// Register module to system
pModuleDef := ISystemBase.regModule(pAdsInfo:=ADR(sC_Ads_Info), pMapInfo:=ADR(sMappingInfo));
IF pModuleDef = 0 THEN RETURN; END_IF

// Command / Status interface
PRG_SYSTEMBASE.getSystemStatusInterface(iSystemStatus=>iSystemStatus);
PRG_SYSTEMBASE.getSystemCmdInterface(iSystemCmd=>iSystemCmd);

// Let the sleep be handled by the library
iSystemCmd.registerPucSleepInterface(pCmd_Sleep:=ADR(sADS_Machine[1].sI_Sleep),
                                     pCmd_WakeUp:=ADR(sADS_Machine[1].sI_WakeUp));

// Get Task cycle information
Fb_GetCurTskIndx();
tskL_ActTaskInfo := _TaskInfo[FB_GetCurTskIndx.index];
lL_TaskCycleTime := UDINT_TO_REAL(tskL_ActTaskInfo.CycleTime) / 10_000_000.0;

(* -- Messages ----------------------------------------------------------------------------------*)
initMsg();


(*************************************************************************************************)
(*Function Blocks Init*)
(*************************************************************************************************)
(*Cleaning station*)
(*Module 1*)
sADS_CleanProcess[1].aO_Name                  := 'Clean Process M2';
sADS_CleanProcess[1].bO_AxisProcessMovingVisible := FALSE;
//Clean unit
sADS_CleanAxis[1].aO_Name                     := 'M2: CU-Axis [mm]';
sADS_CleanAxis[1].sO_AxisPosition.fC_Min      := 0;    (*Value is used for display of axes at PUC*)
sADS_CleanAxis[1].sO_AxisPosition.fC_Max      := 586.0;
fb_CleaningCU[1].pC_MsgInterface              := ADR(sADS_CleanAxis[1].sO_Message);
fb_CleaningCU[1].iC_BlockId                   := eMa_BLK_CLEANAXIS;
fb_CleaningCU[1].fB_Axis.fI_Tolerance         := 0.001;
fb_CleaningCU[1].fB_Axis.fI_PosControllerGain := 5;
fb_CleaningCU[1].fB_Axis.fI_Axis_Scaling      := (0.1512 * 1/10);
fb_CleaningCU[1].fB_Axis.fI_SetPositionValue  := -0.01;				(*Reference sensor is at -10mm*)
fb_CleaningCU[1].fB_Axis.fI_EncoderScaling    := 1048576			(*262.144 * 4*);

//Clean head
sADS_CleanAxis[2].aO_Name                     := 'M2: CH-Axis [mm]';
sADS_CleanAxis[2].sO_AxisPosition.fC_Min      := -1;
sADS_CleanAxis[2].sO_AxisPosition.fC_Max      := 400.0;
fb_CleaningCH[1].pC_MsgInterface              := ADR(sADS_CleanAxis[2].sO_Message);
fb_CleaningCH[1].iC_BlockId                   := eMa_BLK_CLEANAXIS;
fb_CleaningCH[1].fB_Axis.fI_Tolerance         := 0.001;
fb_CleaningCH[1].fB_Axis.fI_PosControllerGain := 5;
fb_CleaningCH[1].fB_Axis.fI_Axis_Scaling      := (0.010 * 1/10);
fb_CleaningCH[1].fB_Axis.fI_SetPositionValue  := -0.001;      (*Reference sensor is at -1mm*)
fb_CleaningCH[1].fB_Axis.fI_EncoderScaling    := 1048576			(*262.144 * 4*);

//Print unit
sADS_CleanAxis[3].aO_Name                     := 'M2: PU-Axis [mm]';
sADS_CleanAxis[3].sO_AxisPosition.fC_Min      := 0.5;  (********(Köbi) Korrektur 0.5 statt 1 *)
sADS_CleanAxis[3].sO_AxisPosition.fC_Max      := 250;
fb_CleaningPU[1].pC_MsgInterface              := ADR(sADS_CleanAxis[3].sO_Message);
fb_CleaningPU[1].iC_BlockId                   := eMa_BLK_CLEANAXIS;
fb_CleaningPU[1].fB_Axis.fI_Tolerance         := 0.0001;
fb_CleaningPU[1].fB_Axis.fI_PosControllerGain := 10;
fb_CleaningPU[1].fB_Axis.fI_Axis_Scaling      := 0.001; (******(Köbi) Korrektur Ration 0.001 statt ...*) //0.016 / 50 * 3;	(*Steigung Spindel / Übersetzung * Winkelgetriebe*)
fb_CleaningPU[1].fB_Axis.fI_SetPositionValue  := 0.010;           (*Calibrate manually at 10mm*)
fb_CleaningPU[1].fB_Axis.fI_EncoderScaling    := 1048576			(*65536*);

//Ink interface
sADS_CleanAxis[4].sO_AxisPosition.fC_Min      := 0;     (*Dummy*)
sADS_CleanAxis[4].sO_AxisPosition.fC_Max      := 1000;  (*Dummy*)


(*Module 2*)
sADS_CleanProcess[2].aO_Name                  := 'Clean Process M3';
sADS_CleanProcess[2].bO_AxisProcessMovingVisible := FALSE;
//Clean unit
sADS_CleanAxis[5].aO_Name                     := 'M3: CU-Axis [mm]';
sADS_CleanAxis[5].sO_AxisPosition.fC_Min      := 0;    (*Value is used for display of axes at PUC*)
sADS_CleanAxis[5].sO_AxisPosition.fC_Max      := 586.0;
fb_CleaningCU[2].pC_MsgInterface              := ADR(sADS_CleanAxis[5].sO_Message);
fb_CleaningCU[2].iC_BlockId                   := eMa_BLK_CLEANAXIS;
fb_CleaningCU[2].fB_Axis.fI_Tolerance         := 0.001;
fb_CleaningCU[2].fB_Axis.fI_PosControllerGain := 5;
fb_CleaningCU[2].fB_Axis.fI_Axis_Scaling      := (0.1512 * 1/10);
fb_CleaningCU[2].fB_Axis.fI_SetPositionValue  := -0.01;				(*Reference sensor is at -10mm*)
fb_CleaningCU[2].fB_Axis.fI_EncoderScaling    := 1048576			(*262.144 * 4*);

//Clean head
sADS_CleanAxis[6].aO_Name                     := 'M3: CH-Axis [mm]';
sADS_CleanAxis[6].sO_AxisPosition.fC_Min      := -1;
sADS_CleanAxis[6].sO_AxisPosition.fC_Max      := 400.0;
fb_CleaningCH[2].pC_MsgInterface              := ADR(sADS_CleanAxis[6].sO_Message);
fb_CleaningCH[2].iC_BlockId                   := eMa_BLK_CLEANAXIS;
fb_CleaningCH[2].fB_Axis.fI_Tolerance         := 0.001;
fb_CleaningCH[2].fB_Axis.fI_PosControllerGain := 5;
fb_CleaningCH[2].fB_Axis.fI_Axis_Scaling      := (0.010 * 1/10);
fb_CleaningCH[2].fB_Axis.fI_SetPositionValue  := -0.001;      (*Reference sensor is at -1mm*)
fb_CleaningCH[2].fB_Axis.fI_EncoderScaling    := 1048576			(*262.144 * 4*);

//Print unit
sADS_CleanAxis[7].aO_Name                     := 'M3: PU-Axis [mm]';
sADS_CleanAxis[7].sO_AxisPosition.fC_Min      := 0.5;  (********(Köbi) Korrektur 0.5 statt 1 *)
sADS_CleanAxis[7].sO_AxisPosition.fC_Max      := 250;
fb_CleaningPU[2].pC_MsgInterface              := ADR(sADS_CleanAxis[7].sO_Message);
fb_CleaningPU[2].iC_BlockId                   := eMa_BLK_CLEANAXIS;
fb_CleaningPU[2].fB_Axis.fI_Tolerance         := 0.0001;
fb_CleaningPU[2].fB_Axis.fI_PosControllerGain := 10;
fb_CleaningPU[2].fB_Axis.fI_Axis_Scaling      := 0.001; (******(Köbi) Korrektur Ration 0.001 statt ...*) //0.016 / 50 * 3;	(*Steigung Spindel / Übersetzung * Winkelgetriebe*)
fb_CleaningPU[2].fB_Axis.fI_SetPositionValue  := 0.010;            (*Calibrate manually at 10mm*)
fb_CleaningPU[2].fB_Axis.fI_EncoderScaling    := 1048576			(*65536*);

//Ink interface
sADS_CleanAxis[8].sO_AxisPosition.fC_Min      := 0;     (*Dummy*)
sADS_CleanAxis[8].sO_AxisPosition.fC_Max      := 1000;  (*Dummy*)

//Link reference to machine base
//X: clean unit
//Y: clean head
//Z: print unit
FOR iL_Counter := 1 TO iCMa_NB_Cp DO
  fb_CleanProcess     [iL_Counter].I_MachineStatus := fb_Machine;
  fb_CleaningCU       [iL_Counter].I_MachineStatus := fb_Machine;
  fb_CleaningPU       [iL_Counter].I_MachineStatus := fb_Machine;
  fb_CleaningCH       [iL_Counter].I_MachineStatus := fb_Machine;
  fb_CleaningValvePump[iL_Counter].I_MachineStatus := fb_Machine;
  
  //Init blocks
  fb_CleanProcess[iL_Counter].pC_MsgInterface := ADR(sADS_CleanProcess[iL_Counter].sO_Message);
  fb_CleanProcess[iL_Counter].iC_BlockId      := eMa_BLK_CLEANPROC;
  
  fb_CleanProcess     [iL_Counter].mInit();
  fb_CleaningCU       [iL_Counter].mInit();
  fb_CleaningPU       [iL_Counter].mInit();
  fb_CleaningCH       [iL_Counter].mInit();
  fb_CleaningValvePump[iL_Counter].mInit();
  
  //Register cleaning devices
  fb_CleanProcess[iL_Counter].mRegisterDevice(fb_CleaningCU[iL_Counter]);
  fb_CleanProcess[iL_Counter].mRegisterDevice(fb_CleaningPU[iL_Counter]);
  fb_CleanProcess[iL_Counter].mRegisterDevice(fb_CleaningCH[iL_Counter]);
  fb_CleanProcess[iL_Counter].mRegisterDevice(fb_CleaningValvePump[iL_Counter]);

  fb_MotionInterlock[iL_Counter].fCCU_SafePosition[1]      := 0.005;
  fb_MotionInterlock[iL_Counter].fCCU_SafePosition[2]      := 0.584;
  fb_MotionInterlock[iL_Counter].fCCU_SafePosition[3]      := 0.586;
  fb_MotionInterlock[iL_Counter].fCPU_SafePosition[1]      := 0.160;
  fb_MotionInterlock[iL_Counter].fCPU_SafePosition[2]      := 0.165;
  fb_MotionInterlock[iL_Counter].fCCU_CleaningPosition     := 0.584;
  fb_MotionInterlock[iL_Counter].fCCU_Tolerance            := 0.002;
  fb_MotionInterlock[iL_Counter].fCPU_Tolerance            := 0.0005;
END_FOR;

(* -- Mapping -----------------------------------------------------------------------------------*)
Mapping();

(* -- Recipe ------------------------------------------------------------------------------------*)
pFbRecipeMngr := PRG_SYSTEMBASE.registerRecipe(
  aI_RecipePath           := CONCAT(aC_PlcConfigPath, aC_PlcRecipeSubPath),
  aI_RecipeDefinitionName := sC_Ads_Info.aType  (*is set in Mapping*)
);

(* -- BlockId saving ----------------------------------------------------------------------------*)
PRG_SYSTEMBASE.fbBlockIdSave.registerModule(
  aI_StoragePath := CONCAT(aC_PlcConfigPath, aC_PlcBlockIdSubPath),
  pI_Ads_Info    := ADR(sC_Ads_Info)
);

bL_RemVar_Init := TRUE;    (* Write variables by remanent variables *)
RemVar();

// init finished
bO_InitOk :=  TRUE;
END_METHOD

METHOD PRIVATE initMsg

(*Machine messaging*)
sL_MsgConfigMachine[1].bI_Enable                  := TRUE;
sL_MsgConfigMachine[1].pI_FbMsgHandler            := ADR(fb_MachineMsgHandler[1]);

fb_MachineMsgHandler[1].pI_MsgQueue               := ADR(fb_MsgQueueMachine[1]);

fb_MsgQueueMachine[1].pI_MsgInterface             := ADR(sADS_Machine[1].sO_Message);
fb_MsgQueueMachine[1].cI_MaxElement               := 5;

FOR iL_Counter := 1 TO iCMa_NB_MSG DO
  fb_MachineMsg[1, iL_Counter].pI_MsgConfig       := ADR(sL_MsgConfigMachine[1]);
  fb_MachineMsg[1, iL_Counter].iI_MsgLocation     := 1;
END_FOR;

fb_MachineMsg[1, 1].iI_MsgNumber                  := eCMa_EMERGENCY_STOP_ACTIVE;
fb_MachineMsg[1, 2].iI_MsgNumber                  := eCMa_MACHINE_DISABLED;
fb_MachineMsg[1, 3].iI_MsgNumber                  := eCMa_MACHINE_COMM_ERR;
fb_MachineMsg[1, 4].iI_MsgNumber                  := eCMa_SLEEP_MODE_ACTIVE;
fb_MachineMsg[1, 5].iI_MsgNumber                  := eCMa_TEMPERATURE_MONITORING;
fb_MachineMsg[1, 6].iI_MsgNumber                  := eCMa_STOR_TANKS_DISABLED;
fb_MachineMsg[1, 7].iI_MsgNumber                  := eCMa_INK_WC_STATE_ERROR;
fb_MachineMsg[1, 8].iI_MsgNumber                  := eCMa_PRINT_WC_STATE_ERROR;
fb_MachineMsg[1, 9].iI_MsgNumber                  := eCMa_MACHINE_WC_STATE_ERROR;
fb_MachineMsg[1,10].iI_MsgNumber                  := eCMa_TCPIP_COMM_ERROR;
fb_MachineMsg[1,11].iI_MsgNumber                  := eCIk_CLEANER_CONTAINER_LEVEL_EMPTY;
fb_MachineMsg[1,12].iI_MsgNumber                  := eCIk_REFUSE_CONTAINER_LEVEL_FULL;
fb_MachineMsg[1,13].iI_MsgNumber                  := eCMa_AXIS_ERROR_X_PNEUMATIC;
fb_MachineMsg[1,14].iI_MsgNumber                  := eCMa_WATCH_CIRCUIT_BREAKER;
fb_MachineMsg[1,15].iI_MsgNumber                  := eCMa_COVER_INLET;
fb_MachineMsg[1,16].iI_MsgNumber                  := eCMa_COVER_OUTLET;
fb_MachineMsg[1,17].iI_MsgNumber                  := eCMa_WATCH_CABINET_TEMP;
fb_MachineMsg[1,18].iI_MsgNumber                  := eCMa_WATCH_SEPARATOR_NIVEAU;
fb_MachineMsg[1,19].iI_MsgNumber                  := eCMa_AXIS_SAFETY_ACCEPTANCE;
fb_MachineMsg[1,20].iI_MsgNumber                  := eCMa_DRIFT_CONTR_ERROR;
fb_MachineMsg[1,21].iI_MsgNumber                  := eCIk_CLEAN_START_MISSING;
fb_MachineMsg[1,22].iI_MsgNumber                  := eCMa_RECIPE_LOADED;
fb_MachineMsg[1,23].iI_MsgNumber                  := eCMa_AXIS_ERROR_Z_PNEUMATIC;
fb_MachineMsg[1,24].iI_MsgNumber                  := eCMa_CLEANER_TANK_INFO;
fb_MachineMsg[1,25].iI_MsgNumber                  := eCMa_MAX_SPEED_EXCEEDED;
fb_MachineMsg[1,26].iI_MsgNumber                  := eCMa_IMAGE_DEPTH_INCORRECT;
fb_MachineMsg[1,27].iI_MsgNumber                  := eCMa_EXHAUST_SYSTEM_WARNING;
fb_MachineMsg[1,28].iI_MsgNumber                  := eCMa_EXHAUST_SYSTEM_ERROR;
fb_MachineMsg[1,29].iI_MsgNumber                  := eCMa_EXHAUST_SYSTEM_MALFUNCTION;
fb_MachineMsg[1,30].iI_MsgNumber                  := eCMa_CLEANER_TANK_FILLING;
fb_MachineMsg[1,31].iI_MsgNumber                  := eCMa_SEPARATOR_LEVEL_REACHED;
END_METHOD

ACTION Mapping:
(*************************************************************************************************)
(*ADS blocks mapping definition*)
(*************************************************************************************************)
(*mapping of each block with his parents, type and index*)
(*Cleaning process -> root*)
sL_BLK_CP[1].iPMaps[1]	:=	FC_ADD_MAP(eSys_BLK_ROOT, 1);
sL_BLK_CP[2].iPMaps[1]	:=	FC_ADD_MAP(eSys_BLK_ROOT, 1);

(*Axis -> Cleaning process*)
sL_BLK_AX[1].iPMaps[1]	:=	FC_ADD_MAP(eMa_BLK_CLEANPROC, 1);
sL_BLK_AX[2].iPMaps[1]	:=	FC_ADD_MAP(eMa_BLK_CLEANPROC, 1);
sL_BLK_AX[3].iPMaps[1]	:=	FC_ADD_MAP(eMa_BLK_CLEANPROC, 1);
sL_BLK_AX[5].iPMaps[1]	:=	FC_ADD_MAP(eMa_BLK_CLEANPROC, 2);
sL_BLK_AX[6].iPMaps[1]	:=	FC_ADD_MAP(eMa_BLK_CLEANPROC, 2);
sL_BLK_AX[7].iPMaps[1]	:=	FC_ADD_MAP(eMa_BLK_CLEANPROC, 2);

(*Machine -> root*)
sL_BLK_MA[1].iPMaps[1]	:=	FC_ADD_MAP(eSys_BLK_ROOT, 1);


(*************************************************************************************************)
(*ADS blocks configuration & information*)
(*************************************************************************************************)
sC_Ads_Info.bReady   := FALSE;
sC_Ads_Info.aType    := 'PRG_MACHINE';
sC_Ads_Info.iVersion := 010000;			(*1.0.0*)
sC_Ads_Info.iType    := eMOD_MACHINE;

sMappingInfo.init(lModId:=TO_UINT(eMOD_MACHINE)); 
sMappingInfo.addBlkAry( iAdsBlockType := TO_UINT(eMa_BLK_MACHINE)  , aAdsBlockName := 'sADS_Machine'     , iAdsBlockVersion:= INT_TO_UINT(sADS_Machine     [1].iO_Version), iNbrBlocks := SIZEOF(sL_BLK_MA) / SIZEOF(sL_BLK_MA[1]), pBlockArray := ADR(sL_BLK_MA));
sMappingInfo.addBlkAry( iAdsBlockType := TO_UINT(eMa_BLK_CLEANPROC), aAdsBlockName := 'sADS_CleanProcess', iAdsBlockVersion:= INT_TO_UINT(sADS_CleanProcess[1].iO_Version), iNbrBlocks := SIZEOF(sL_BLK_CP) / SIZEOF(sL_BLK_CP[1]), pBlockArray := ADR(sL_BLK_CP));
sMappingInfo.addBlkAry( iAdsBlockType := TO_UINT(eMa_BLK_CLEANAXIS), aAdsBlockName := 'sADS_CleanAxis'   , iAdsBlockVersion:= INT_TO_UINT(sADS_CleanAxis   [1].iO_Version), iNbrBlocks := SIZEOF(sL_BLK_AX) / SIZEOF(sL_BLK_AX[1]), pBlockArray := ADR(sL_BLK_AX));
sMappingInfo.bReady := TRUE;
END_ACTION

ACTION RemVar:
(*************************************************************************************************)
(********************************* READING REMANENT VARIABLES ************************************)
(*************************************************************************************************)
IF bL_RemVar_Init THEN

  (*load initial values if pattern was invalid*)
  IF sR_RemVar_M.aL_Pattern <> 16#ABCD THEN

    lL_ToleranceLenPx              := 5;      (*[px]*)

    (*Recipe: load and write*)
    IF pFbRecipeMngr <> 0 THEN
      pFbRecipeMngr^.mWriteRecipe('');
      bL_RecipeValuesLoadedMachine := TRUE;
    END_IF

  ELSE

    sR_RemVar_M.aL_Pattern := sR_RemVar_M.aL_Pattern;  (*TODO remove dummy code*)

    lL_ToleranceLenPx      := sR_RemVar_M.lR_ToleranceLenPx;

  END_IF


  bL_RemVar_Init := FALSE;

(*************************************************************************************************)
(********************************* WRITING REMANENT VARIABLES ************************************)
(*************************************************************************************************)
ELSE

(*GENERAL*)
(*************************************************************************************************)
  sR_RemVar_M.aL_Pattern := 16#ABCD;


  sR_RemVar_M.lR_ToleranceLenPx    := lL_ToleranceLenPx;
END_IF;
END_ACTION

ACTION Simulate:

IF bL_SimInputs THEN
  bIKp_SeparatorNiveau_Ok[1] := TRUE;
  bIKp_SeparatorNiveau_Ok[2] := TRUE;
  (*
  fb_CleaningPU[1].fI_PositionService := 210;
  fb_CleaningPU[2].fI_PositionService := 210;
  fb_CleaningPU[1].fI_PositionWait    := 55;
  fb_CleaningPU[2].fI_PositionWait    := 55;
  fb_CleaningPU[1].fI_PositionPrint   := 1;
  fb_CleaningPU[2].fI_PositionPrint   := 1;
  *)
END_IF

fbMachineComm.bSimEnable := bSimulation;
END_ACTION

METHOD updateSleepLock
sADS_Machine[1].sI_Sleep.bO_CommandCanEx := sADS_Machine[1].sI_Sleep.bO_CommandCanEx AND bAllowSleepFromMachine;
END_METHOD

END_PROGRAM

// ---- POUs/Products/Machine/CleaningStation/FB_CleaningMotorAxisCU.TcPOU
FUNCTION_BLOCK FB_CleaningMotorAxisCU EXTENDS FB_CleanDevice
VAR_INPUT
  bI_SafeToMove                        : BOOL;
  
  //Limit switches
  bI_ReferenceSensor            AT %I* : BOOL;  (*Physical sensor feedback reference position*)
  
  //Inputs from EL7201 Terminal
  wI_StatusWord                 AT %I* : UINT; (*Status word: 6041:0*)
  lI_EncoderValue               AT %I* : DINT; (*Encoder value*)
  bI_DeviceOnline               AT %I* : BOOL; (*Check link to device*)
  
  fB_Axis                              : FB_EL7201;    //Axis controller
  
  //References
  pC_MsgInterface                      : POINTER TO ST_ADS_MSG_IF;
  iC_BlockId                           : INT;
END_VAR

VAR_OUTPUT
  //Outputs to EL7201 Terminal
  wO_ControlWord                AT %Q* : UINT;                         (*Control word:  6040:0*)
  iO_TargetVelocity             AT %Q* : DINT;                         (*Target velocity:  60FF:0*)
END_VAR

VAR
  //Limit switches
  bL_ReferenceSensor                   : BOOL;  (*Negated sensor feedback reference position*)

  fb_TonDeviceOnline                   : TON;
	bIDp_DeviceReset                     : BOOL := FALSE;
	fb_RTrigDeviceReset                  : R_TRIG;

  bL_SafeRunningCondition              : BOOL;
  bL_SafeMoveNeg                       : BOOL;
  bL_SafeMovePos                       : BOOL;
  bL_memRefSensor                      : BOOL;
  bL_FirstRun                          : BOOL := TRUE;

  fL_ManualMoveTolerance               : REAL := 0.001;
  
  bL_InPosCappClean                    : BOOL;
  bL_InPosPark                         : BOOL;
  
  wL_ErrorCode                         : WORD;
  
  (*Messaging*)
  fB_MsgQueue                          : FB_MSG_QUEUE;
  fB_MsgHandler                        : FB_MSG_HANDLER;
  sL_MsgConfig                         : ST_MSG_CONFIG;
  fB_Msg                               : ARRAY [1..iC_NUM_MSG] OF FB_MESSAGE;
END_VAR

VAR PERSISTENT
  fI_PositionCappingClean              : REAL;           (*[mm]*)
  fI_PositionPark                      : REAL;           (*[mm]*)
  fI_PositionTolerance                 : REAL := 0.001;  (*[m]*)
  sI_SpeedDef                          : ST_SPEEDS;  (*Speed defs [mm/s]*)
END_VAR

VAR CONSTANT
  iC_NUM_MSG                           : INT  := 1;
END_VAR

//Limit switches for internal use
bL_ReferenceSensor := NOT bI_ReferenceSensor;

(*----------------------------------------------------------------------------------------------------------------------------------------------- *)
(*Running Conditions for Cleaning Unit  *)
(*----------------------------------------------------------------------------------------------------------------------------------------------- *)
IF I_MachineStatus.pSafetyOk AND I_MachineStatus.pMachineReady AND (wL_ErrorCode = 0 OR wL_ErrorCode.5)THEN  (*Dont check limit switch here*)
  bL_SafeRunningCondition := TRUE;
ELSE
  bL_SafeRunningCondition := FALSE;
END_IF;

bL_SafeMoveNeg := bL_SafeRunningCondition AND NOT bL_ReferenceSensor AND bI_SafeToMove;
bL_SafeMovePos := bL_SafeRunningCondition AND bI_SafeToMove;

(*Because the WcState sets an error for on cycle, we use this timer to check if the bus is down.*)
fb_TonDeviceOnline(IN := bI_DeviceOnline, PT := T#20MS);
fb_RTrigDeviceReset(CLK := bIDp_DeviceReset);
IF fb_TonDeviceOnline.Q OR fb_RTrigDeviceReset.Q THEN
  bL_RefKnown    := FALSE;        (*Reset Reference when link to device is lost, e.g. when machine power off*)
	wL_ErrorCode.9 := TRUE;
END_IF;

(*----------------------------------------------------------------------------------------------------------------------------------------------- *)
(*Position detection*)
(*----------------------------------------------------------------------------------------------------------------------------------------------- *)
IF     fB_Axis.fO_ActualPosition >= ((fI_PositionCappingClean / 1000) - fI_PositionTolerance)
   AND fB_Axis.fO_ActualPosition <= ((fI_PositionCappingClean / 1000) + fI_PositionTolerance)
THEN
  bL_InPosCappClean := TRUE;
  bL_InPosPark      := FALSE;
ELSIF  fB_Axis.fO_ActualPosition >= ((fI_PositionPark / 1000) - fI_PositionTolerance)
   AND fB_Axis.fO_ActualPosition <= ((fI_PositionPark / 1000) + fI_PositionTolerance)
THEN
  bL_InPosCappClean := FALSE;
  bL_InPosPark      := TRUE;
ELSE
  bL_InPosCappClean := FALSE;
  bL_InPosPark      := FALSE;
END_IF;


(*----------------------------------------------------------------------------------------------------------------------------------------------- *)
(* Axis control  *)
(*----------------------------------------------------------------------------------------------------------------------------------------------- *)
fB_Axis.bI_RegActive := bL_SafeRunningCondition AND NOT bL_Error; //Activate controller
fB_Axis.bI_EStop     := I_MachineStatus.pSafetyOk;                //negative logic for bI_EStop

fB_Axis(wI_StatusWord := wI_StatusWord ,lI_EncoderValue := lI_EncoderValue);

fB_Axis.bI_FaultReset := FALSE;

wO_ControlWord    := fB_Axis.wO_ControlWord;
iO_TargetVelocity := fB_Axis.iO_TargetVelocity;


(*----------------------------------------------------------------------------------------------------------------------------------------------- *)
(* Supervision  *)
(*----------------------------------------------------------------------------------------------------------------------------------------------- *)
(*
TODO: Supervisor
tL_TimerSurv.PT := T#3S;
tL_TimerSurv();
tL_TimerSensor.PT := T#105s  ;  (* 1meter at 10mm*)
tL_TimerSensor();*)

IF bL_FirstRun THEN
  bL_FirstRun     := FALSE;
  bL_memRefSensor := bL_ReferenceSensor;
END_IF;

(*----------------------------------------------------------------------------------------------------------------------- *)
(*--------------------------------- Fault Diagnosis and Management  ----------------------------------------------------- *)
(*----------------------------------------------------------------------------------------------------------------------- *)
mErrorHandling();

(*----------------------------------------------------------------------------------------------------------------------- *)
(* Messaging                                                                                                              *)
(*----------------------------------------------------------------------------------------------------------------------- *)
fB_MsgHandler();
fB_Msg[1](bI_Status := bL_Error);
fB_MsgQueue();

METHOD mAckError 
VAR_INPUT
END_VAR
wL_ErrorCode := 0;
mErrorHandling();
fB_Axis.bI_FaultReset := TRUE;
END_METHOD

METHOD mCapping : BOOL
VAR_INPUT
  iI_Step    : INT;
  bI_ExitCap : BOOL;
END_VAR
//Abort: Stop whereever axis is and return
IF bL_AbortReq THEN
  fB_Axis.bI_MoveEnable := FALSE;
  bL_Busy  := FALSE;
  bL_Ready := TRUE;

  RETURN;
END_IF

//Normal operation
bL_Ready := FALSE;
CASE iI_Step OF
	0: //Init - Check if axis is not activated, restore safety
    fB_Axis.bI_MoveEnable := FALSE;
		bL_Busy := FALSE;

  1: //Wait for PU axis to lift
    fB_Axis.bI_MoveEnable   := FALSE;
    bL_Busy                 := FALSE;
    
  2: //Wait for CU axis to move in
    mAckError();
    fB_Axis.fI_TargetPosition := (fI_PositionCappingClean / 1000);
    fB_Axis.fI_SpeedLimit     := sI_SpeedDef.fP_PlaceSpeed / 1000;
    
    IF bL_InPosCappClean THEN
      fB_Axis.bI_MoveEnable := FALSE;
      bL_Busy               := FALSE;
      bL_Ready              := TRUE;  //Operation complete
    ELSE
      fB_Axis.bI_MoveEnable := bL_SafeMovePos;
      bL_Busy               := TRUE;
    END_IF
    
  3: //Move CH to park positiom 
    fB_Axis.bI_MoveEnable   := FALSE;
    bL_Busy                 := FALSE;
    
  4: //Wait for PU axis to lower
    fB_Axis.bI_MoveEnable   := FALSE;
    bL_Busy                 := FALSE;
    
	5: //End - Do nothing, capping process active
    mAckError();
		bL_Busy  := FALSE;
    bL_Ready := TRUE;  //Operation complete

	ELSE
		bL_Busy  := FALSE;		
    bL_Ready := TRUE;  //Operation complete
END_CASE
END_METHOD

METHOD mCleaning : BOOL
VAR_INPUT
  iI_Step : INT;
END_VAR
//Abort: Stop whereever axis is and return
IF bL_AbortReq THEN
  fB_Axis.bI_MoveEnable := FALSE;
  bL_Busy  := FALSE;
  bL_Ready := TRUE;

  RETURN;
END_IF

//Normal operation
bL_Ready := FALSE;
CASE iI_Step OF
  0: //Init - Check if axis is not activated, restore safety
    bL_Busy := FALSE;

  1: //Wait for PU axis to lift
    fB_Axis.bI_MoveEnable   := FALSE;
    bL_Busy                 := FALSE;
    
  2: //Wait for CU axis to move in
    mAckError();
    fB_Axis.fI_TargetPosition := (fI_PositionCappingClean / 1000);
    fB_Axis.fI_SpeedLimit     := sI_SpeedDef.fP_PlaceSpeed / 1000;
    
    IF bL_InPosCappClean THEN
      fB_Axis.bI_MoveEnable := FALSE;
      bL_Busy               := FALSE;
      bL_Ready              := TRUE;  //Operation complete
    ELSE
      fB_Axis.bI_MoveEnable := bL_SafeMovePos;
      bL_Busy               := TRUE;
    END_IF
    
  3: //Wait for PU axis to lower
    fB_Axis.bI_MoveEnable   := FALSE;
    bL_Busy                 := FALSE;
    
  4: //Ensure CH axis is at starting position
    fB_Axis.bI_MoveEnable   := FALSE;
    bL_Busy                 := FALSE;
    
  5: //Move CH to clean start position
    fB_Axis.bI_MoveEnable   := FALSE;
    bL_Busy                 := FALSE;

  6: //Wait until cleaning equipment ready
    fB_Axis.bI_MoveEnable   := FALSE;
    bL_Busy                 := FALSE;
    
  7: //Cleaning
    fB_Axis.bI_MoveEnable   := FALSE;
    bL_Busy                 := FALSE;  
    
  8: //Wait until cleaning equipment ready
    fB_Axis.bI_MoveEnable   := FALSE;
    bL_Busy                 := FALSE;
    
  9: //Move CH to end position
    fB_Axis.bI_MoveEnable   := FALSE;
    bL_Busy                 := FALSE;  
    
  10: //Wait for PU axis to lift
    fB_Axis.bI_MoveEnable   := FALSE;
    bL_Busy                 := FALSE;  
  
  11: //Move CH back to start 
    fB_Axis.bI_MoveEnable   := FALSE;
    bL_Busy                 := FALSE;  

  12: //Wait for PU axis to lower
    fB_Axis.bI_MoveEnable   := FALSE;
    bL_Busy                 := FALSE;
    
  13: //End
    fB_Axis.bI_MoveEnable   := FALSE;
    bL_Busy                 := FALSE;  
    bL_Ready                := TRUE;  //Operation complete

  ELSE
    bL_Busy  := FALSE;    
    bL_Ready := TRUE;  //Operation complete
END_CASE
END_METHOD

METHOD PRIVATE mErrorHandling
VAR_INPUT
END_VAR
fB_Msg[1].bI_Status := FALSE;

IF (sI_SpeedDef.fP_PlaceSpeed = 0) OR (sI_SpeedDef.fP_WorkSpeed = 0) OR (sI_SpeedDef.fP_ServiceSpeed = 0) THEN	(* Speed Configuration not done *)
	wL_ErrorCode.6 := TRUE;
END_IF;

IF (fI_PositionCappingClean = 0) THEN		(* Position Configuration not done *)
	wL_ErrorCode.7 := TRUE;
END_IF;

IF fB_Axis.eO_EL7201Status = eFault  THEN
	wL_ErrorCode.8 := TRUE;						(* EL7342 module fault *)
	fB_Msg[1].bI_Status := TRUE;
END_IF;


IF wl_ErrorCode = 0 THEN
	bL_Error := FALSE;
ELSE
	bL_Error := TRUE;
END_IF;
END_METHOD

METHOD mErrorRecovery : BOOL
VAR_INPUT
    iI_Step : INT;
END_VAR
//Do nothing
bL_Busy  := FALSE;
bL_Ready := TRUE;
END_METHOD

METHOD mInit
VAR_INPUT
END_VAR
(*Messages*)
sL_MsgConfig.bI_Enable       := TRUE;
sL_MsgConfig.pI_FbMsgHandler := ADR(fB_MsgHandler);
fB_MsgHandler.pI_MsgQueue    := ADR(fB_MsgQueue);
fB_MsgQueue.pI_MsgInterface  := pC_MsgInterface;
fB_MsgQueue.cI_MaxElement    := 5;

fB_Msg[1].iI_MsgLocation     := iC_BlockId;
fB_Msg[1].pI_MsgConfig       := ADR(sL_MsgConfig);
fB_Msg[1].iI_MsgNumber       := eCMa_AxisErrorX;
END_METHOD

METHOD mManuellMove : BOOL
VAR_INPUT
  bI_Do                  : BOOL;
  fI_TargetPosition      : REAL;
  fL_ManualMoveTolerance : REAL;
END_VAR
fB_Axis.fI_SpeedLimit     := sI_SpeedDef.fP_ServiceSpeed / 1000;
fB_Axis.fI_TargetPosition := fI_TargetPosition / 1000;
IF fB_Axis.fI_TargetPosition > fB_Axis.fO_ActualPosition THEN
  fB_Axis.bI_MoveEnable   := bI_Do AND bL_SafeMovePos;
ELSIF fB_Axis.fI_TargetPosition < fB_Axis.fO_ActualPosition THEN
  fB_Axis.bI_MoveEnable   := bI_Do AND bL_SafeMoveNeg;
ELSE
  fB_Axis.bI_MoveEnable   := bI_Do;
END_IF

bL_Busy  := ABS(fB_Axis.fI_TargetPosition - fB_Axis.fO_ActualPosition) > fL_ManualMoveTolerance;
bL_Ready := NOT (ABS(fB_Axis.fI_TargetPosition - fB_Axis.fO_ActualPosition) > fL_ManualMoveTolerance);  //Operation complete
END_METHOD

METHOD mProduction : BOOL
VAR_INPUT
  iI_Step : INT;
END_VAR
//Abort: Stop whereever axis is and return
IF bL_AbortReq THEN
  fB_Axis.bI_MoveEnable := FALSE;
  bL_Busy  := FALSE;
  bL_Ready := TRUE;

  RETURN;
END_IF

//Normal operation
bL_Ready := FALSE;
CASE iI_Step OF
  0: //Init - Check if axis is not activated, restore safety
    bL_Busy := FALSE;

  1: //Wait for PU axis to lift
    fB_Axis.bI_MoveEnable   := FALSE;
    bL_Busy                 := FALSE;
    
  2: //Wait for CU axis to move out
    mAckError();
    fB_Axis.fI_TargetPosition := (fI_PositionPark / 1000);
    fB_Axis.fI_SpeedLimit     := sI_SpeedDef.fP_PlaceSpeed / 1000;
    
    IF bL_InPosPark THEN
      fB_Axis.bI_MoveEnable := FALSE;
      bL_Busy               := FALSE;
      bL_Ready              := TRUE;  //Operation complete
    ELSE
      fB_Axis.bI_MoveEnable := bL_SafeMoveNeg;
      bL_Busy               := TRUE;
    END_IF
    
  3: //Wait for PU axis to lower
    fB_Axis.bI_MoveEnable   := FALSE;
    bL_Busy                 := FALSE;
    
  4: //End
    fB_Axis.bI_MoveEnable := FALSE;
    bL_Busy               := FALSE;  
    bL_Ready              := TRUE;  //Operation complete

  ELSE
    bL_Busy  := FALSE;    
    bL_Ready := TRUE;  //Operation complete
END_CASE
END_METHOD

METHOD mService : BOOL
VAR_INPUT
  iI_Step : INT;
END_VAR
//Abort: Stop whereever axis is and return
IF bL_AbortReq THEN
  fB_Axis.bI_MoveEnable := FALSE;
  bL_Busy  := FALSE;
  bL_Ready := TRUE;

  RETURN;
END_IF

//Normal operation
bL_Ready := FALSE;
CASE iI_Step OF
  0: //Init - Check if axis is not activated, restore safety
    bL_Busy := FALSE;

  1: //Wait for PU axis to lift to ExitCapping
    fB_Axis.bI_MoveEnable   := FALSE;
    bL_Busy                 := FALSE;
    
  2: //Wait for CU axis to move in
    mAckError();
    fB_Axis.fI_TargetPosition := (fI_PositionPark / 1000);
    fB_Axis.fI_SpeedLimit     := sI_SpeedDef.fP_PlaceSpeed / 1000;
    
    IF bL_InPosPark THEN
      fB_Axis.bI_MoveEnable := FALSE;
      bL_Busy               := FALSE;
      bL_Ready              := TRUE;  //Operation complete
    ELSE
      fB_Axis.bI_MoveEnable := bL_SafeMoveNeg;
      bL_Busy               := TRUE;
    END_IF
    
  3: //End
    fB_Axis.bI_MoveEnable := FALSE;
    bL_Busy               := FALSE;  
    bL_Ready              := TRUE;

  ELSE
    bL_Busy  := FALSE;    
    bL_Ready := TRUE;  //Operation complete
END_CASE
END_METHOD

METHOD mStartup : BOOL
VAR_INPUT
  iI_Step : INT;
END_VAR
CASE iI_Step OF
	0: //Init - Check if axis is not activated, restore safety
		bL_Busy := FALSE;

	1: //Wait until other axes in place
		bL_Busy := FALSE;

	2: //Begin - Init CU axis if NOT bL_RefKnown
    bL_Busy  := NOT bL_RefKnown;
    bL_Ready := bL_RefKnown;
    
    fB_Axis.bI_SetPosition := bL_RefKnown;
    
    IF NOT bL_RefKnown THEN  (* if the CU axis hasn't been initialized with Ref Sensor*)
      IF bL_ReferenceSensor AND NOT bL_memRefSensor AND NOT bL_RefKnown THEN
        bL_RefKnown             := TRUE;                      (* When the sensor is activated, Save the correction value*)
        fB_Axis.bI_SetPosition  := TRUE;                      (*Initialize position to preset value*)
        fB_Axis.bI_MoveEnable   := FALSE;
        bL_Ready                := TRUE;
      ELSE
        IF bL_ReferenceSensor AND bL_memRefSensor THEN
          fB_Axis.fI_TargetPosition := fB_Axis.fO_ActualPosition + 0.01;  (*@@@@CONST, change to JOG_NEGATIVE*)
          fB_Axis.fI_SpeedLimit     := sI_SpeedDef.fP_ServiceSpeed / 1000;     (* Start backward motion, the motor will run until Ref Sensor is ON*)
          fB_Axis.bI_MoveEnable     := bL_SafeMovePos;
        ELSE
          fB_Axis.fI_TargetPosition := -100.0;                               (*@@@@CONST, change to JOG_NEGATIVE*)
          fB_Axis.fI_SpeedLimit     := sI_SpeedDef.fP_ServiceSpeed / 1000;  (* Start backward motion, the motor will run until Ref Sensor is ON*)
          fB_Axis.bI_MoveEnable     := bL_SafeMoveNeg;
        END_IF;
      END_IF;
    END_IF;

    bL_memRefSensor := bL_ReferenceSensor;				(* Memorization of the Ref sensor state for edge detection*)

	3,4: //End
		bL_Busy  := FALSE;		
    bL_Ready := TRUE;  //Operation complete

	ELSE
		bL_Busy  := FALSE;		
    bL_Ready := TRUE;  //Operation complete
END_CASE
END_METHOD

{attribute 'monitoring' := 'call'}
PROPERTY pInPosCappingClean : BOOL
GET
pInPosCappingClean := bL_InPosCappClean;
END_GET
END_PROPERTY

{attribute 'monitoring' := 'call'}
PROPERTY pInPosPark : bool
GET
pInPosPark := bL_InPosPark;
END_GET
END_PROPERTY

END_FUNCTION_BLOCK

// ---- POUs/Products/Machine/CleaningStation/FB_CleaningMotorAxisCH.TcPOU
FUNCTION_BLOCK FB_CleaningMotorAxisCH EXTENDS FB_CleanDevice
VAR_INPUT
  bI_SafeToMove                        : BOOL;
  
  //Limit switches
  bI_Sensor_pA                  AT %I* : BOOL;  (*Physical sensor feedback for pA position*)
  bI_Sensor_pB                  AT %I* : BOOL;  (*Physical sensor feedback for pB position*)
  
  //Inputs from EL7201 Terminal
  wI_StatusWord                 AT %I* : UINT; (*Status word: 6041:0*)
  lI_EncoderValue               AT %I* : DINT; (*Encoder value*)
  bI_DeviceOnline               AT %I* : BOOL; (*Check link to device*)
  
  fB_Axis                              : FB_EL7201;    //Axis controller
  
  //References
  pC_MsgInterface                      : POINTER TO ST_ADS_MSG_IF;
  iC_BlockId                           : INT;
END_VAR

VAR_OUTPUT
  //Outputs to EL7201 Terminal
  wO_ControlWord                AT %Q* : UINT;                         (*Control word:  6040:0*)
  iO_TargetVelocity             AT %Q* : DINT;                         (*Target velocity:  60FF:0*)
END_VAR

VAR
  //Limit switches
  bL_Sensor_pA                         : BOOL;  (*Negated sensor feedback for pA position*)
  bL_Sensor_pB                         : BOOL;  (*Negated sensor feedback for pB position*)

  fb_TonDeviceOnline                   : TON;
	bIDp_DeviceReset                     : BOOL := FALSE;
	fb_RTrigDeviceReset                  : R_TRIG;

  bL_SafeRunningCondition              : BOOL;
  bL_SafeMoveNeg                       : BOOL;
  bL_SafeMovePos                       : BOOL;
  bL_memRefSensor                      : BOOL;
  bL_FirstRun                          : BOOL := TRUE;

  bL_InPosA                            : BOOL;
  bL_InPosB                            : BOOL;
  
  wL_ErrorCode                         : WORD;
  
  (*Messaging*)
  fB_MsgQueue                          : FB_MSG_QUEUE;
  fB_MsgHandler                        : FB_MSG_HANDLER;
  sL_MsgConfig                         : ST_MSG_CONFIG;
  fB_Msg                               : ARRAY [1..iC_NUM_MSG] OF FB_MESSAGE;
END_VAR

VAR PERSISTENT
  fI_Position_p1                       : REAL;           (*[mm]*)
  fI_Position_p2                       : REAL;           (*[mm]*)
  fI_Position_A                        : REAL;           (*[mm]*)
  fI_Position_B                        : REAL;           (*[mm]*)
  fI_PositionTolerance                 : REAL := 0.001;  (*[m]*)
  sI_SpeedDef                          : ST_SPEEDS;  (*Speed defs [mm/s]*)
END_VAR

VAR CONSTANT
  iC_NUM_MSG                           : INT  := 1;
END_VAR

//Limit switches for internal use
bL_Sensor_pA := NOT bI_Sensor_pA;
bL_Sensor_pB := FALSE; (*not existing:  NOT bI_Sensor_pB;*)

(*----------------------------------------------------------------------------------------------------------------------------------------------- *)
(*Running Conditions for Cleaning Head  *)
(*----------------------------------------------------------------------------------------------------------------------------------------------- *)
IF bI_SafeToMove AND I_MachineStatus.pSafetyOk AND I_MachineStatus.pMachineReady AND (wL_ErrorCode = 0 OR wL_ErrorCode.5)THEN  (*Dont check limit switch here*)
  bL_SafeRunningCondition := TRUE;
ELSE
  bL_SafeRunningCondition := FALSE;
END_IF;

bL_SafeMoveNeg := bL_SafeRunningCondition AND NOT bL_Sensor_pA;
bL_SafeMovePos := bL_SafeRunningCondition AND NOT bL_Sensor_pB;

(*Because the WcState sets an error for on cycle, we use this timer to check if the bus is down.*)
fb_TonDeviceOnline(IN := bI_DeviceOnline, PT := T#20MS);
fb_RTrigDeviceReset(CLK := bIDp_DeviceReset);
IF fb_TonDeviceOnline.Q OR fb_RTrigDeviceReset.Q THEN
  bL_RefKnown    := FALSE;        (*Reset Reference when link to device is lost, e.g. when machine power off*)
	wL_ErrorCode.9 := TRUE;
END_IF;

(*----------------------------------------------------------------------------------------------------------------------------------------------- *)
(*Position detection*)
(*----------------------------------------------------------------------------------------------------------------------------------------------- *)
IF     (fB_Axis.fO_ActualPosition >= ((fI_Position_A / 1000) - fI_PositionTolerance)
   AND  fB_Axis.fO_ActualPosition <= ((fI_Position_A / 1000) + fI_PositionTolerance)) OR bL_Sensor_pA
THEN
  bL_InPosA := TRUE;
  bL_InPosB := FALSE;
ELSIF  fB_Axis.fO_ActualPosition >= ((fI_Position_B / 1000) - fI_PositionTolerance)
   AND fB_Axis.fO_ActualPosition <= ((fI_Position_B / 1000) + fI_PositionTolerance)
THEN
  bL_InPosA := FALSE;
  bL_InPosB := TRUE;
ELSE
  bL_InPosA := FALSE;
  bL_InPosB := FALSE;
END_IF;


(*----------------------------------------------------------------------------------------------------------------------------------------------- *)
(* Axis control  *)
(*----------------------------------------------------------------------------------------------------------------------------------------------- *)
fB_Axis.bI_RegActive := bL_SafeRunningCondition AND NOT bL_Error; //Activate controller
fB_Axis.bI_EStop     := I_MachineStatus.pSafetyOk;                //negative logic for bI_EStop

fB_Axis(wI_StatusWord := wI_StatusWord ,lI_EncoderValue := lI_EncoderValue);

fB_Axis.bI_FaultReset := FALSE;

wO_ControlWord    := fB_Axis.wO_ControlWord;
iO_TargetVelocity := fB_Axis.iO_TargetVelocity;


(*----------------------------------------------------------------------------------------------------------------------------------------------- *)
(* Supervision  *)
(*----------------------------------------------------------------------------------------------------------------------------------------------- *)
(*
TODO: Supervisor
tL_TimerSurv.PT := T#3S;
tL_TimerSurv();
tL_TimerSensor.PT := T#105s  ;  (* 1meter at 10mm*)
tL_TimerSensor();*)

IF bL_FirstRun THEN
  bL_FirstRun     := FALSE;
  bL_memRefSensor := bL_Sensor_pA;
END_IF;

(*----------------------------------------------------------------------------------------------------------------------- *)
(*--------------------------------- Fault Diagnosis and Management  ----------------------------------------------------- *)
(*----------------------------------------------------------------------------------------------------------------------- *)
mErrorHandling();

(*----------------------------------------------------------------------------------------------------------------------- *)
(* Messaging                                                                                                              *)
(*----------------------------------------------------------------------------------------------------------------------- *)
fB_MsgHandler();
fB_Msg[1](bI_Status := bL_Error);
fB_MsgQueue();

METHOD mAckError 
VAR_INPUT
END_VAR
wL_ErrorCode := 0;
mErrorHandling();
fB_Axis.bI_FaultReset := TRUE;
END_METHOD

METHOD mCapping : BOOL
VAR_INPUT
  iI_Step    : INT;
  bI_ExitCap : BOOL;
END_VAR
//Abort: Stop whereever axis is and return
IF bL_AbortReq THEN
  fB_Axis.bI_MoveEnable := FALSE;
  bL_Busy  := FALSE;
  bL_Ready := TRUE;

  RETURN;
END_IF

//Normal operation
bL_Ready := FALSE;
CASE iI_Step OF
	0: //Init - Check if axis is not activated, restore safety
    fB_Axis.bI_MoveEnable := FALSE;
		bL_Busy := FALSE;

  1: //Wait for PU axis to lift
    fB_Axis.bI_MoveEnable   := FALSE;
    bL_Busy                 := FALSE;
    
  2: //Wait for CU axis to move in
    fB_Axis.bI_MoveEnable   := FALSE;
    bL_Busy                 := FALSE;
    
  3: //Move CH to park positiom 
    fB_Axis.fI_TargetPosition := (fI_Position_A / 1000);
    fB_Axis.fI_SpeedLimit     := sI_SpeedDef.fP_PlaceSpeed / 1000;
    
    IF bL_InPosA THEN //Target reached
      fB_Axis.bI_MoveEnable := FALSE;
      bL_Busy               := FALSE;
      bL_Ready              := TRUE;  //Operation complete
    ELSE
      fB_Axis.bI_MoveEnable := bL_SafeMoveNeg;
      bL_Busy               := TRUE;
    END_IF

  4: //Wait for PU axis to lower
    fB_Axis.bI_MoveEnable   := FALSE;
    bL_Busy                 := FALSE;
    
	5: //End - Do nothing, capping process active
    mAckError();
		bL_Busy  := FALSE;
    bL_Ready := TRUE;  //Operation complete

	ELSE
		bL_Busy  := FALSE;		
    bL_Ready := TRUE;  //Operation complete
END_CASE
END_METHOD

METHOD mCleaning : BOOL
VAR_INPUT
  iI_Step : INT;
END_VAR
//Abort: Stop whereever axis is and return
IF bL_AbortReq THEN
  bL_Busy:=FALSE;
  fB_Axis.bI_MoveEnable:=FALSE;
  bL_Ready := TRUE;
  RETURN;
END_IF

//Normal operation
bL_Ready := FALSE;
CASE iI_Step OF
  0: //Init - Check if axis is not activated, restore safety
    bL_Busy := FALSE;

  1: //Wait for PU axis to lift
    fB_Axis.bI_MoveEnable   := FALSE;
    bL_Busy                 := FALSE;
    
  2: //Wait for CU axis to move in
    fB_Axis.bI_MoveEnable   := FALSE;
    bL_Busy                 := FALSE;
    
  3: //Wait for PU axis to lower
    fB_Axis.bI_MoveEnable   := FALSE;
    bL_Busy                 := FALSE;
    
  4: //Ensure CH axis is at starting position
    mAckError();
    fB_Axis.fI_TargetPosition := (fI_Position_A / 1000);
    fB_Axis.fI_SpeedLimit     := sI_SpeedDef.fP_PlaceSpeed / 1000;
    
    IF bL_InPosA THEN
      fB_Axis.bI_MoveEnable := FALSE;
      bL_Busy               := FALSE;
      bL_Ready              := TRUE;  //Operation complete
    ELSE
      fB_Axis.bI_MoveEnable := TRUE;
      bL_Busy               := TRUE;
    END_IF
    
  5: //Move CH to clean start position
    fB_Axis.fI_TargetPosition := (fI_Position_p1 / 1000);
    fB_Axis.fI_SpeedLimit     := sI_SpeedDef.fP_PlaceSpeed / 1000;
    
    IF bL_Sensor_pB OR bL_InPosB THEN //Error
      ; //TODO
    ELSIF fB_Axis.fO_ActualPosition >= (fI_Position_p1 / 1000) THEN //Target reached
      fB_Axis.bI_MoveEnable := FALSE;
      bL_Busy               := FALSE;
      bL_Ready              := TRUE;  //Operation complete
    ELSE
      fB_Axis.bI_MoveEnable := bL_SafeMovePos;
      bL_Busy               := TRUE;
    END_IF

  6: //Wait until cleaning equipment ready
    fB_Axis.bI_MoveEnable   := FALSE;
    bL_Busy                 := FALSE;
    
  7: //Cleaning
    fB_Axis.fI_TargetPosition := (fI_Position_p2 / 1000);
    fB_Axis.fI_SpeedLimit     := sI_SpeedDef.fP_WorkSpeed / 1000;
    
    IF bL_Sensor_pB OR bL_InPosB THEN //Error
      ; //TODO
    ELSIF fB_Axis.fO_ActualPosition >= (fI_Position_p2 / 1000) THEN //Target reached
      fB_Axis.bI_MoveEnable := FALSE;
      bL_Busy               := FALSE;
      bL_Ready              := TRUE;  //Operation complete
    ELSE
      fB_Axis.bI_MoveEnable := bL_SafeMovePos;
      bL_Busy               := TRUE;
    END_IF
    
  8: //Wait until cleaning equipment ready
    fB_Axis.bI_MoveEnable   := FALSE;
    bL_Busy                 := FALSE;
    
  9: //Move CH to end position
    fB_Axis.fI_TargetPosition := (fI_Position_B / 1000);
    fB_Axis.fI_SpeedLimit     := sI_SpeedDef.fP_PlaceSpeed / 1000;
    
    IF bL_InPosB THEN //Target reached
      fB_Axis.bI_MoveEnable := FALSE;
      bL_Busy               := FALSE;
      bL_Ready              := TRUE;  //Operation complete
    ELSE
      fB_Axis.bI_MoveEnable := bL_SafeMovePos;
      bL_Busy               := TRUE;
    END_IF
    
  10: //Wait for PU axis to lift
    fB_Axis.bI_MoveEnable := FALSE;
    bL_Busy               := FALSE;  
  
  11: //Move CH back to start 
    fB_Axis.fI_TargetPosition := (fI_Position_A / 1000);
    fB_Axis.fI_SpeedLimit     := sI_SpeedDef.fP_PlaceSpeed / 1000;
    
    IF bL_InPosA THEN //Target reached
      fB_Axis.bI_MoveEnable := FALSE;
      bL_Busy               := FALSE;
      bL_Ready              := TRUE;  //Operation complete
    ELSE
      fB_Axis.bI_MoveEnable := bL_SafeMoveNeg;
      bL_Busy               := TRUE;
    END_IF

  12: //Wait for PU axis to lower
    fB_Axis.bI_MoveEnable   := FALSE;
    bL_Busy                 := FALSE;
    
  13: //End
    fB_Axis.bI_MoveEnable := FALSE;
    bL_Busy               := FALSE;  
    bL_Ready              := TRUE;  //Operation complete

  ELSE
    bL_Busy  := FALSE;    
    bL_Ready := TRUE;  //Operation complete
END_CASE
END_METHOD

METHOD PRIVATE mErrorHandling
VAR_INPUT
END_VAR
fB_Msg[1].bI_Status := FALSE;

IF (bL_Sensor_pB AND bL_Sensor_pA) THEN			(* Sensor Fault : pB and pA can't be active at the same time *)
	wL_ErrorCode.2 := TRUE ;
END_IF;

IF (sI_SpeedDef.fP_PlaceSpeed=0) OR  (sI_SpeedDef.fP_WorkSpeed=0) OR (sI_SpeedDef.fP_ServiceSpeed=0) THEN	(* Speed Configuration not done *)
	wL_Errorcode.6 := TRUE;
END_IF;

IF (fI_Position_p1=0) OR (fI_Position_p2=0) THEN		(* Position Configuration not done *)
	wL_ErrorCode.7 := TRUE;
END_IF;

IF fB_Axis.eO_EL7201Status = eFault  THEN
	wL_ErrorCode.8 := TRUE;						(* EL7342 module fault *)
	fB_Msg[1].bI_Status := TRUE;
END_IF;


IF wl_ErrorCode = 0 THEN
	bL_Error := FALSE;
ELSE
	bL_Error := TRUE;
END_IF;
END_METHOD

METHOD mErrorRecovery : BOOL
VAR_INPUT
    iI_Step : INT;
END_VAR
//Do nothing
bL_Busy := FALSE;
bL_Ready := TRUE;
END_METHOD

METHOD mInit
VAR_INPUT
END_VAR
	(*Messages*)
	sL_MsgConfig.bI_Enable       := TRUE;
	sL_MsgConfig.pI_FbMsgHandler := ADR(fB_MsgHandler);
	fB_MsgHandler.pI_MsgQueue    := ADR(fB_MsgQueue);
	fB_MsgQueue.pI_MsgInterface  := pC_MsgInterface;
	fB_MsgQueue.cI_MaxElement    := 5;

	fB_Msg[1].iI_MsgLocation     := iC_BlockId;
	fB_Msg[1].pI_MsgConfig       := ADR(sL_MsgConfig);
	fB_Msg[1].iI_MsgNumber       := eCMa_AxisErrorY;
END_METHOD

METHOD mManuellMove : BOOL
VAR_INPUT
  bI_Do                  : BOOL;
  fI_TargetPosition      : REAL;
  fL_ManualMoveTolerance : REAL;
END_VAR
fB_Axis.fI_SpeedLimit     := sI_SpeedDef.fP_ServiceSpeed / 1000;
fB_Axis.fI_TargetPosition := fI_TargetPosition / 1000;
IF fB_Axis.fI_TargetPosition > fB_Axis.fO_ActualPosition THEN
  fB_Axis.bI_MoveEnable   := bI_Do AND bL_SafeMovePos;
ELSIF fB_Axis.fI_TargetPosition < fB_Axis.fO_ActualPosition THEN
  fB_Axis.bI_MoveEnable   := bI_Do AND bL_SafeMoveNeg;
ELSE
  fB_Axis.bI_MoveEnable   := bI_Do;
END_IF

bL_Busy  := ABS(fB_Axis.fI_TargetPosition - fB_Axis.fO_ActualPosition) > fL_ManualMoveTolerance;
bL_Ready := NOT (ABS(fB_Axis.fI_TargetPosition - fB_Axis.fO_ActualPosition) > fL_ManualMoveTolerance);  //Operation complete
END_METHOD

METHOD mProduction : BOOL
VAR_INPUT
  iI_Step : INT;
END_VAR
//Nothing to do
fB_Axis.bI_MoveEnable := FALSE;
bL_Busy  := FALSE;
bL_Ready := TRUE;
END_METHOD

METHOD mService : BOOL
VAR_INPUT
  iI_Step : INT;
END_VAR
//Nothing to do
fB_Axis.bI_MoveEnable := FALSE;
bL_Busy  := FALSE;
bL_Ready := TRUE;
END_METHOD

METHOD mStartup : BOOL
VAR_INPUT
  iI_Step : INT;
END_VAR
CASE iI_Step OF
	0: //Init - Check if axis is not activated, restore safety
		bL_Busy := FALSE;

	1,2: //Wait until other axes in place
		bL_Busy := FALSE;

	3: //Begin - Init CH axis if NOT bL_RefKnown
    bL_Busy  := NOT bL_RefKnown;
    bL_Ready := bL_RefKnown;
    
    fB_Axis.bI_SetPosition := bL_RefKnown;
    
    IF NOT bL_RefKnown THEN  (* if the Y axis hasn't been initialized with Ref Sensor*)
      IF bL_Sensor_pA AND NOT bL_memRefSensor AND NOT bL_RefKnown THEN
        bL_RefKnown             := TRUE;                      (* When the sensor is activated, Save the correction value*)
        fB_Axis.bI_SetPosition  := TRUE;                      (*Initialize position to preset value*)
        fB_Axis.bI_MoveEnable   := FALSE;
        bL_Ready                := TRUE;
      ELSE
        IF bL_Sensor_pA AND bL_memRefSensor THEN
          fB_Axis.fI_TargetPosition := fB_Axis.fO_ActualPosition + 0.01;  (*@@@@CONST, change to JOG_NEGATIVE*)
          fB_Axis.fI_SpeedLimit     := sI_SpeedDef.fP_ServiceSpeed / 1000;     (* Start backward motion, the motor will run until Ref Sensor is ON*)
          fB_Axis.bI_MoveEnable     := bL_SafeMovePos;
        ELSIF bL_Sensor_pB THEN (*Security check if sensor malfunction:*)
          ; //Error
        ELSE
          fB_Axis.fI_TargetPosition := -100.0;                               (*@@@@CONST, change to JOG_NEGATIVE*)
          fB_Axis.fI_SpeedLimit     := (sI_SpeedDef.fP_ServiceSpeed * 0.1) / 1000;  (* Start backward motion, the motor will run until Ref Sensor is ON*)
          fB_Axis.bI_MoveEnable     := bL_SafeMoveNeg;
        END_IF;
      END_IF;
    END_IF;

    bL_memRefSensor := bL_Sensor_pA;				(* Memorization of the Ref sensor state for edge detection*)

	4: //End
		bL_Busy  := FALSE;		
    bL_Ready := TRUE;  //Operation complete

	ELSE
		bL_Busy  := FALSE;		
    bL_Ready := TRUE;  //Operation complete
END_CASE
END_METHOD

{attribute 'monitoring' := 'call'}
PROPERTY pInPosA : bool
GET
pInPosA := bL_InPosA;
END_GET
END_PROPERTY

{attribute 'monitoring' := 'call'}
PROPERTY pInPosB : bool
GET
pInPosB := bL_InPosB;
END_GET
END_PROPERTY

END_FUNCTION_BLOCK

// ---- POUs/Products/Machine/CleaningStation/FB_CleaningMotorAxisPU.TcPOU
FUNCTION_BLOCK FB_CleaningMotorAxisPU EXTENDS FB_CleanDevice
VAR_INPUT
  bI_SafeToMove                        : BOOL;
	fI_SheetThickness                    : REAL := 0.000; (*Sheet thickness (Production Mode) [mm]*)
  
  //Limit switches
  bI_SensorTop                  AT %I* : BOOL;  (*Physical sensor feedback for top position*)
  bI_SensorBottom               AT %I* : BOOL;  (*Physical sensor feedback for bottom position*)
  
  //Inputs from EL7201 Terminal
  wI_StatusWord                 AT %I* : UINT; (*Status word: 6041:0*)
  lI_EncoderValue               AT %I* : DINT; (*Encoder value*)
  bI_DeviceOnline               AT %I* : BOOL; (*Check link to device*)
  
  fB_Axis                              : FB_EL7201;    //Axis controller
  
  //References
  pC_MsgInterface                      : POINTER TO ST_ADS_MSG_IF;
  iC_BlockId                           : INT;
END_VAR

VAR_OUTPUT
  //Outputs to EL7201 Terminal
  wO_ControlWord                AT %Q* : UINT;                         (*Control word:  6040:0*)
  iO_TargetVelocity             AT %Q* : DINT;                         (*Target velocity:  60FF:0*)
END_VAR

VAR
  fb_TonDeviceOnline                   : TON;
	bIDp_DeviceReset                     : BOOL := FALSE;
	fb_RTrigDeviceReset                  : R_TRIG;
  fb_RFTrigPrintEnabled                : RF_TRIG;

  bL_DriveToWaitPos                    : BOOL;
  bL_DriveToPrintPos                   : BOOL;


  bL_SafeRunningCondition              : BOOL;
  bL_SafeMoveNeg                       : BOOL;
  bL_SafeMovePos                       : BOOL;
  bL_FirstRun                          : BOOL := TRUE;

  fL_PrintPosition                     : REAL;  (*[m]*)
  fL_PrintPositionMM                   : REAL;  (*[mm]*)
  bL_InPosService                      : BOOL;
  bL_InPosClean1                       : BOOL;
  bL_InPosClean2                       : BOOL;
  bL_InPosWait                         : BOOL;
  bL_InPosPrint                        : BOOL;
  bL_HigherPosWait                     : BOOL;
  bL_HigherPosC1                       : BOOL;
  
  bL_MemSensorTop                      : BOOL;
  bL_MemSensorBottom                   : BOOL;
  wL_ErrorCode                         : WORD;
  
  (*Messaging*)
  fB_MsgQueue                          : FB_MSG_QUEUE;
  fB_MsgHandler                        : FB_MSG_HANDLER;
  sL_MsgConfig                         : ST_MSG_CONFIG;
  fB_Msg                               : ARRAY [1..iC_NUM_MSG] OF FB_MESSAGE;
END_VAR

VAR PERSISTENT
  fI_PositionService                   : REAL;  (*[mm]*)
  fI_PositionWait                      : REAL;  (*[mm]*)
  fI_PositionClean1                    : REAL;  (*[mm]*)
  fI_PositionClean2                    : REAL;  (*[mm]*)
  fI_PositionPrint                     : REAL;  (*[mm]*)
  fL_SetPositionValue                  : REAL := 10;      (*[mm]*)
  fI_PositionTolerance                 : REAL := 0.0001;  (*[m]*)
  fI_PositionTolerance2                : REAL := 0.005;   (*[m]*)
  sI_SpeedDef                          : ST_SPEEDS;  (*Speed defs [mm/s]*)
END_VAR

VAR CONSTANT
  iC_NUM_MSG                           : INT  := 1;
END_VAR

(*----------------------------------------------------------------------------------------------------------------------------------------------- *)
(*Running Conditions for Cleaning Head  *)
(*----------------------------------------------------------------------------------------------------------------------------------------------- *)
IF I_MachineStatus.pSafetyOk AND I_MachineStatus.pMachineReady AND (wL_ErrorCode = 0 OR wL_ErrorCode.5)THEN  (*Dont check limit switch here*)
  bL_SafeRunningCondition := TRUE;
ELSE
  bL_SafeRunningCondition := FALSE;
END_IF;

bL_SafeMoveNeg := bL_SafeRunningCondition AND bI_SensorBottom AND bI_SafeToMove;
bL_SafeMovePos := bL_SafeRunningCondition AND bI_SensorTop;

(*Because the WcState sets an error for on cycle, we use this timer to check if the bus is down.*)
fb_TonDeviceOnline(IN := bI_DeviceOnline, PT := T#20MS);
fb_RTrigDeviceReset(CLK := bIDp_DeviceReset);
IF fb_TonDeviceOnline.Q OR fb_RTrigDeviceReset.Q THEN
  bL_RefKnown    := FALSE;        (*Reset Reference when link to device is lost, e.g. when machine power off*)
	wL_ErrorCode.9 := TRUE;
END_IF;

(*----------------------------------------------------------------------------------------------------------------------------------------------- *)
(*Position detection*)
(*----------------------------------------------------------------------------------------------------------------------------------------------- *)
fL_PrintPositionMM := fI_PositionPrint + fI_SheetThickness;
fL_PrintPosition   := (fL_PrintPositionMM / 1000);

IF     fB_Axis.fO_ActualPosition >= ((fI_PositionWait / 1000) - (fI_PositionTolerance / 1000))
   AND fB_Axis.fO_ActualPosition <= ((fI_PositionWait / 1000) + (fI_PositionTolerance / 1000))
THEN
  bL_InPosService := FALSE;
  bL_InPosClean1  := FALSE;
  bL_InPosClean2  := FALSE;
  bL_InPosWait    := TRUE;
  bL_InPosPrint   := FALSE;
ELSIF  fB_Axis.fO_ActualPosition >= (fL_PrintPosition - fI_PositionTolerance)
   AND fB_Axis.fO_ActualPosition <= (fL_PrintPosition + fI_PositionTolerance)
THEN
  bL_InPosService := FALSE;
  bL_InPosClean1  := FALSE;
  bL_InPosClean2  := FALSE;
  bL_InPosWait    := FALSE;
  bL_InPosPrint   := TRUE;
ELSIF  fB_Axis.fO_ActualPosition >= ((fI_PositionService / 1000) - fI_PositionTolerance)
   AND fB_Axis.fO_ActualPosition <= ((fI_PositionService / 1000) + fI_PositionTolerance)
THEN
  bL_InPosService := TRUE;
  bL_InPosClean1  := FALSE;
  bL_InPosClean2  := FALSE;
  bL_InPosWait    := FALSE;
  bL_InPosPrint   := FALSE;
ELSIF  fB_Axis.fO_ActualPosition >= ((fI_PositionClean1 / 1000) - fI_PositionTolerance)
   AND fB_Axis.fO_ActualPosition <= ((fI_PositionClean1 / 1000) + fI_PositionTolerance)
THEN
  bL_InPosService := FALSE;
  bL_InPosClean1  := TRUE;
  bL_InPosClean2  := FALSE;
  bL_InPosWait    := FALSE;
  bL_InPosPrint   := FALSE;
ELSIF  fB_Axis.fO_ActualPosition >= ((fI_PositionClean2 / 1000) - fI_PositionTolerance)
   AND fB_Axis.fO_ActualPosition <= ((fI_PositionClean2 / 1000) + fI_PositionTolerance)
THEN
  bL_InPosService := FALSE;
  bL_InPosClean1  := FALSE;
  bL_InPosClean2  := TRUE;
  bL_InPosWait    := FALSE;
  bL_InPosPrint   := FALSE;
ELSE
  bL_InPosService := FALSE;
  bL_InPosClean1  := FALSE;
  bL_InPosClean2  := FALSE;
  bL_InPosWait    := FALSE;
  bL_InPosPrint   := FALSE;
END_IF;
bL_HigherPosWait := fB_Axis.fO_ActualPosition >= ((fI_PositionWait   / 1000) + fI_PositionTolerance2);
bL_HigherPosC1   := fB_Axis.fO_ActualPosition >= ((fI_PositionClean1 / 1000));

(*----------------------------------------------------------------------------------------------------------------------------------------------- *)
(* Axis control  *)
(*----------------------------------------------------------------------------------------------------------------------------------------------- *)
fB_Axis.bI_RegActive        := bL_SafeRunningCondition AND NOT bL_Error; //Activate controller
fB_Axis.bI_EStop            := I_MachineStatus.pSafetyOk;                //negative logic for bI_EStop
fB_Axis.fI_SetPositionValue := fL_SetPositionValue / 1000;

fB_Axis(wI_StatusWord := wI_StatusWord ,lI_EncoderValue := lI_EncoderValue);

fB_Axis.bI_FaultReset := FALSE;

wO_ControlWord    := fB_Axis.wO_ControlWord;
iO_TargetVelocity := fB_Axis.iO_TargetVelocity;

IF fB_Axis.fL_OffsetEncoder > 0 THEN
	bL_RefKnown := TRUE;
ELSE
	bL_RefKnown := FALSE;
END_IF;


(*----------------------------------------------------------------------------------------------------------------------------------------------- *)
(* Supervision  *)
(*----------------------------------------------------------------------------------------------------------------------------------------------- *)
(*
TODO: Supervisor
tL_TimerSurv.PT := T#3S;
tL_TimerSurv();
tL_TimerSensor.PT := T#105s  ;  (* 1meter at 10mm*)
tL_TimerSensor();*)

IF bL_FirstRun THEN
  bL_FirstRun     := FALSE;
END_IF;

(*----------------------------------------------------------------------------------------------------------------------- *)
(*--------------------------------- Fault Diagnosis and Management  ----------------------------------------------------- *)
(*----------------------------------------------------------------------------------------------------------------------- *)
mErrorHandling();

(*----------------------------------------------------------------------------------------------------------------------- *)
(* Messaging                                                                                                              *)
(*----------------------------------------------------------------------------------------------------------------------- *)
fB_MsgHandler();
fB_Msg[1](bI_Status := bL_Error);
fB_MsgQueue();

METHOD mAckError 
VAR_INPUT
END_VAR
wL_ErrorCode := 0;
mErrorHandling();
fB_Axis.bI_FaultReset := TRUE;
END_METHOD

METHOD mCapping : BOOL
VAR_INPUT
  iI_Step    : INT;
  bI_ExitCap : BOOL;
END_VAR
//Abort: Stop whereever axis is and return
IF bL_AbortReq THEN
  fB_Axis.bI_MoveEnable := FALSE;
  bL_Busy  := FALSE;
  bL_Ready := TRUE;

  RETURN;
END_IF

//Normal operation
bL_Ready := FALSE;
CASE iI_Step OF
	0: //Init - Check if axis is not activated, restore safety
    fB_Axis.bI_MoveEnable := FALSE;
		bL_Busy               := FALSE;

  1: //Wait for PU axis to lift
    mAckError();
    fB_Axis.fI_TargetPosition := (fI_PositionClean1 / 1000);
    fB_Axis.fI_SpeedLimit     := sI_SpeedDef.fP_PlaceSpeed / 1000;
    
    IF bL_InPosClean1 THEN
      fB_Axis.bI_MoveEnable := FALSE;
      bL_Busy               := FALSE;
      bL_Ready              := TRUE;  //Operation complete
    ELSE
      fB_Axis.bI_MoveEnable := bL_SafeMovePos;
      bL_Busy               := TRUE;
    END_IF
    
  2: //Wait for CU axis to move in
    fB_Axis.bI_MoveEnable   := FALSE;
    bL_Busy                 := FALSE;
    
  3: //Move CH to park positiom 
    fB_Axis.bI_MoveEnable   := FALSE;
    bL_Busy                 := FALSE;
    
  4: //Wait for PU axis to lower
    mAckError();
    IF NOT bI_ExitCap THEN
      fB_Axis.fI_TargetPosition := (fI_PositionClean2 / 1000);
      fB_Axis.fI_SpeedLimit     := sI_SpeedDef.fP_PlaceSpeed / 1000;
      
      IF bL_InPosClean2 THEN
        fB_Axis.bI_MoveEnable := FALSE;
        bL_Busy               := FALSE;
        bL_Ready              := TRUE;  //Operation complete
      ELSE
        fB_Axis.bI_MoveEnable := bL_SafeMoveNeg;
        bL_Busy               := TRUE;
      END_IF
    ELSE
      fB_Axis.bI_MoveEnable := FALSE;
      bL_Busy               := FALSE;
    END_IF
    
	5: //End - Do nothing, capping process active
    mAckError();
		bL_Busy  := FALSE;
    bL_Ready := TRUE;  //Operation complete

	ELSE
		bL_Busy  := FALSE;		
    bL_Ready := TRUE;  //Operation complete
END_CASE
END_METHOD

METHOD mCleaning : BOOL
VAR_INPUT
  iI_Step : INT;
END_VAR
//Abort: Stop whereever axis is and return
IF bL_AbortReq THEN
  fB_Axis.bI_MoveEnable := FALSE;
  bL_Busy  := FALSE;
  bL_Ready := TRUE;

  RETURN;
END_IF

//Normal operation
bL_Ready := FALSE;
CASE iI_Step OF
  0: //Init - Check if axis is not activated, restore safety
    bL_Busy := FALSE;

  1: //Wait for PU axis to lift
    mAckError();
    fB_Axis.fI_TargetPosition := (fI_PositionClean1 / 1000);
    fB_Axis.fI_SpeedLimit     := sI_SpeedDef.fP_PlaceSpeed / 1000;
    
    IF bL_InPosClean1 THEN
      fB_Axis.bI_MoveEnable := FALSE;
      bL_Busy               := FALSE;
      bL_Ready              := TRUE;  //Operation complete
    ELSE
      fB_Axis.bI_MoveEnable := bL_SafeMovePos;
      bL_Busy               := TRUE;
    END_IF
    
  2: //Wait for CU axis to move in
    fB_Axis.bI_MoveEnable   := FALSE;
    bL_Busy                 := FALSE;
    
  3: //Wait for PU axis to lower
    mAckError();
    fB_Axis.fI_TargetPosition := (fI_PositionClean2 / 1000);
    fB_Axis.fI_SpeedLimit     := sI_SpeedDef.fP_PlaceSpeed / 1000;
    
    IF bL_InPosClean2 THEN
      fB_Axis.bI_MoveEnable := FALSE;
      bL_Busy               := FALSE;
      bL_Ready              := TRUE;  //Operation complete
    ELSE
      fB_Axis.bI_MoveEnable := bL_SafeMoveNeg;
      bL_Busy               := TRUE;
    END_IF
    
  4: //Ensure CH axis is at starting position
    fB_Axis.bI_MoveEnable   := FALSE;
    bL_Busy                 := FALSE;
    
  5: //Move CH to clean start position
    fB_Axis.bI_MoveEnable   := FALSE;
    bL_Busy                 := FALSE;

  6: //Wait until cleaning equipment ready
    fB_Axis.bI_MoveEnable   := FALSE;
    bL_Busy                 := FALSE;
    
  7: //Cleaning
    fB_Axis.bI_MoveEnable   := FALSE;
    bL_Busy                 := FALSE;  
    
  8: //Wait until cleaning equipment ready
    fB_Axis.bI_MoveEnable   := FALSE;
    bL_Busy                 := FALSE;
    
  9: //Move CH to end position
    fB_Axis.bI_MoveEnable   := FALSE;
    bL_Busy                 := FALSE;  
    
  10: //Wait for PU axis to lift
    mAckError();
    fB_Axis.fI_TargetPosition := (fI_PositionClean1 / 1000);
    fB_Axis.fI_SpeedLimit     := sI_SpeedDef.fP_PlaceSpeed / 1000;
    
    IF bL_InPosClean1 THEN
      fB_Axis.bI_MoveEnable := FALSE;
      bL_Busy               := FALSE;
      bL_Ready              := TRUE;  //Operation complete
    ELSE
      fB_Axis.bI_MoveEnable := bL_SafeMovePos;
      bL_Busy               := TRUE;
    END_IF
  
  11: //Move CH back to start 
    fB_Axis.bI_MoveEnable   := FALSE;
    bL_Busy                 := FALSE;  

  12: //Wait for PU axis to lower
    mAckError();
    fB_Axis.fI_TargetPosition := (fI_PositionClean2 / 1000);
    fB_Axis.fI_SpeedLimit     := sI_SpeedDef.fP_PlaceSpeed / 1000;
    
    IF bL_InPosClean2 THEN
      fB_Axis.bI_MoveEnable := FALSE;
      bL_Busy               := FALSE;
      bL_Ready              := TRUE;  //Operation complete
    ELSE
      fB_Axis.bI_MoveEnable := bL_SafeMoveNeg;
      bL_Busy               := TRUE;
    END_IF
    
  13: //End
    fB_Axis.bI_MoveEnable   := FALSE;
    bL_Busy                 := FALSE;  
    bL_Ready                := TRUE;  //Operation complete
  
  ELSE
    bL_Busy  := FALSE;    
    bL_Ready := TRUE;  //Operation complete
END_CASE
END_METHOD

METHOD PRIVATE mErrorHandling
VAR_INPUT
END_VAR
fB_Msg[1].bI_Status := FALSE;

IF NOT bL_RefKnown THEN
	wL_ErrorCode.1 := TRUE;						(* Axis has lost its value *)
END_IF;

IF (NOT bI_SensorTop AND NOT bI_SensorBottom) THEN      (* Sensor Fault : SensorTop and SensorBottom can't be active at the same time *)
	wL_ErrorCode.2 := TRUE;
END_IF;

IF (NOT bI_SensorTop AND bL_MemSensorTop) THEN          (* Safety Fault : Limit Switch Top activated *)
	wL_ErrorCode.3 := TRUE;
END_IF;
bL_MemSensorTop := bI_SensorTop;

IF (NOT bI_SensorBottom AND bL_MemSensorBottom) THEN    (* Safety Fault : Limit Switch Bottom activated *)
	wL_ErrorCode.4 := TRUE;
END_IF;
bL_MemSensorBottom := bI_SensorBottom;

IF (sI_SpeedDef.fP_PlaceSpeed=0) OR  (sI_SpeedDef.fP_WorkSpeed=0) OR (sI_SpeedDef.fP_ServiceSpeed=0) THEN	(* Speed Configuration not done *)
	wL_Errorcode.6 := TRUE;
END_IF;

IF (fI_PositionService = 0) OR (fI_PositionWait = 0) OR (fI_PositionClean1 = 0) OR (fI_PositionClean2 = 0) THEN		(* Position Configuration not done *)
	wL_ErrorCode.7 := TRUE;
END_IF;

IF fB_Axis.eO_EL7201Status = eFault  THEN
	wL_ErrorCode.8 := TRUE;						(* EL7342 module fault *)
	fB_Msg[1].bI_Status := TRUE;
END_IF;


IF wl_ErrorCode = 0 THEN
	bL_Error := FALSE;
ELSE
	bL_Error := TRUE;
END_IF;
END_METHOD

METHOD mErrorRecovery : BOOL
VAR_INPUT
    iI_Step : INT;
END_VAR
//Do nothing
bL_Busy  := FALSE;
bL_Ready := TRUE;
END_METHOD

METHOD mInit
VAR_INPUT
END_VAR
	(*Messages*)
	sL_MsgConfig.bI_Enable       := TRUE;
	sL_MsgConfig.pI_FbMsgHandler := ADR(fB_MsgHandler);
	fB_MsgHandler.pI_MsgQueue    := ADR(fB_MsgQueue);
	fB_MsgQueue.pI_MsgInterface  := pC_MsgInterface;
	fB_MsgQueue.cI_MaxElement    := 5;

	fB_Msg[1].iI_MsgLocation     := iC_BlockId;
	fB_Msg[1].pI_MsgConfig       := ADR(sL_MsgConfig);
	fB_Msg[1].iI_MsgNumber       := eCMa_AxisErrorZ;
END_METHOD

METHOD mManuellMove : BOOL
VAR_INPUT
  bI_Do                  : BOOL;
  fI_TargetPosition      : REAL;
  fL_ManualMoveTolerance : REAL;
END_VAR
IF fB_Axis.fO_ActualPosition < (fI_PositionWait / 1000) THEN
  fB_Axis.fI_SpeedLimit   := sI_SpeedDef.fP_WorkSpeed / 1000;
ELSE
  fB_Axis.fI_SpeedLimit   := sI_SpeedDef.fP_ServiceSpeed / 1000;
END_IF
fB_Axis.fI_TargetPosition := fI_TargetPosition / 1000;
IF fB_Axis.fI_TargetPosition > fB_Axis.fO_ActualPosition THEN
  fB_Axis.bI_MoveEnable   := bI_Do AND bL_SafeMovePos;
ELSIF fB_Axis.fI_TargetPosition < fB_Axis.fO_ActualPosition THEN
  fB_Axis.bI_MoveEnable   := bI_Do AND bL_SafeMoveNeg;
ELSE
  fB_Axis.bI_MoveEnable   := bI_Do;
END_IF

bL_Busy  := ABS(fB_Axis.fI_TargetPosition - fB_Axis.fO_ActualPosition) > fL_ManualMoveTolerance;
bL_Ready := NOT (ABS(fB_Axis.fI_TargetPosition - fB_Axis.fO_ActualPosition) > fL_ManualMoveTolerance);  //Operation complete
END_METHOD

METHOD mPrintPos : BOOL
VAR_INPUT
  bI_PrintEnabled        : BOOL;
  bI_PrintFinsihed       : BOOL;
END_VAR

VAR
  bDriveToWaitPos        : BOOL;
  bDriveToPrintPos       : BOOL;
END_VAR
fb_RFTrigPrintEnabled(CLK := bI_PrintEnabled);
IF fb_RFTrigPrintEnabled.RT THEN bL_DriveToPrintPos := TRUE; bL_DriveToWaitPos  := FALSE; END_IF
IF fb_RFTrigPrintEnabled.FT THEN bL_DriveToWaitPos  := TRUE; bL_DriveToPrintPos := FALSE; END_IF

IF NOT pHigherPosWait AND bL_Ready THEN
  //IF fb_RFTrigPrintEnabled.RT THEN bL_DriveToPrintPos := TRUE; END_IF
  IF bL_DriveToPrintPos THEN
    fB_Axis.fI_TargetPosition := (fL_PrintPosition);
    fB_Axis.fI_SpeedLimit     := sI_SpeedDef.fP_WorkSpeed / 1000;
    
    IF bL_InPosPrint THEN
      fB_Axis.bI_MoveEnable := FALSE;
      bL_Busy               := FALSE;
      bL_DriveToPrintPos    := FALSE;
      bL_Ready              := TRUE;  //Operation complete
    ELSE
      fB_Axis.bI_MoveEnable := bL_SafeMoveNeg;
      bL_Busy               := TRUE;
    END_IF
  END_IF

  //IF fb_RFTrigPrintEnabled.FT THEN bL_bDriveToWaitPos := TRUE; END_IF
  IF bL_DriveToWaitPos AND bI_PrintFinsihed THEN
    fB_Axis.fI_TargetPosition := (fI_PositionWait / 1000);
    fB_Axis.fI_SpeedLimit     := sI_SpeedDef.fP_PlaceSpeed / 1000;
    
    IF bL_InPosWait THEN
      fB_Axis.bI_MoveEnable := FALSE;
      bL_Busy               := FALSE;
      bL_DriveToWaitPos     := FALSE;
      bL_Ready              := TRUE;  //Operation complete
    ELSE
      fB_Axis.bI_MoveEnable := bL_SafeMovePos;
      bL_Busy               := TRUE;
    END_IF
  END_IF
END_IF
END_METHOD

METHOD mProduction : BOOL
VAR_INPUT
  iI_Step : INT;
END_VAR
//Abort: Stop whereever axis is and return
IF bL_AbortReq THEN
  fB_Axis.bI_MoveEnable := FALSE;
  bL_Busy  := FALSE;
  bL_Ready := TRUE;

  RETURN;
END_IF

//Normal operation
bL_Ready := FALSE;
CASE iI_Step OF
  0: //Init - Check if axis is not activated, restore safety
    bL_Busy := FALSE;

  1: //Wait for PU axis to lift
    mAckError();
    fB_Axis.fI_TargetPosition := (fI_PositionClean1 / 1000);
    fB_Axis.fI_SpeedLimit     := sI_SpeedDef.fP_PlaceSpeed / 1000;
    
    IF bL_InPosClean1 THEN
      fB_Axis.bI_MoveEnable := FALSE;
      bL_Busy               := FALSE;
      bL_Ready              := TRUE;  //Operation complete
    ELSE
      fB_Axis.bI_MoveEnable := bL_SafeMovePos;
      bL_Busy               := TRUE;
    END_IF
    
  2: //Wait for CU axis to move out
    fB_Axis.bI_MoveEnable   := FALSE;
    bL_Busy                 := FALSE;
    
  3: //Wait for PU axis to lower
    mAckError();
    fB_Axis.fI_TargetPosition := (fI_PositionWait / 1000);
    fB_Axis.fI_SpeedLimit     := sI_SpeedDef.fP_PlaceSpeed / 1000;
    
    IF bL_InPosWait THEN
      fB_Axis.bI_MoveEnable := FALSE;
      bL_Busy               := FALSE;
      bL_Ready              := TRUE;  //Operation complete
    ELSE
      fB_Axis.bI_MoveEnable := bL_SafeMoveNeg;
      bL_Busy               := TRUE;
    END_IF
    
  4: //End
    fB_Axis.bI_MoveEnable := FALSE;
    bL_Busy               := FALSE;  
    bL_Ready              := TRUE;  //Operation complete

  ELSE
    bL_Busy  := FALSE;    
    bL_Ready := TRUE;  //Operation complete
END_CASE
END_METHOD

METHOD mService : BOOL
VAR_INPUT
  iI_Step : INT;
END_VAR
//Abort: Stop whereever axis is and return
IF bL_AbortReq THEN
  fB_Axis.bI_MoveEnable := FALSE;
  bL_Busy  := FALSE;
  bL_Ready := TRUE;

  RETURN;
END_IF

//Normal operation
bL_Ready := FALSE;
CASE iI_Step OF
  0: //Init - Check if axis is not activated, restore safety
    bL_Busy := FALSE;

  1: //Wait for PU axis to lift to ExitCapping
    mAckError();
    fB_Axis.fI_TargetPosition := (fI_PositionClean1 / 1000);
    fB_Axis.fI_SpeedLimit     := sI_SpeedDef.fP_PlaceSpeed / 1000;
    
    IF bL_InPosClean1 THEN
      fB_Axis.bI_MoveEnable := FALSE;
      bL_Busy               := FALSE;
    ELSE
      fB_Axis.bI_MoveEnable := bL_SafeMovePos;
      bL_Busy               := TRUE;
    END_IF
        
  2: //Wait for PU to reach Service (CU moves out)
    mAckError();
    fB_Axis.fI_TargetPosition := (fI_PositionService / 1000);
    fB_Axis.fI_SpeedLimit     := sI_SpeedDef.fP_PlaceSpeed / 1000;
    
    IF bL_InPosService THEN
      fB_Axis.bI_MoveEnable := FALSE;
      bL_Busy               := FALSE;
      bL_Ready              := TRUE;  //Operation complete
    ELSE
      fB_Axis.bI_MoveEnable := bL_SafeMovePos;
      bL_Busy               := TRUE;
    END_IF
    
  3: //End
    fB_Axis.bI_MoveEnable := FALSE;
    bL_Busy               := FALSE; 
    bL_Ready              := TRUE; 
  
  ELSE
    bL_Busy  := FALSE;    
    bL_Ready := TRUE;  //Operation complete
END_CASE
END_METHOD

METHOD mStartup : BOOL
VAR_INPUT
  iI_Step : INT;
END_VAR
CASE iI_Step OF
	0: //Init - Check if axis is not activated, restore safety
		bL_Busy := FALSE;

  1: //Wait for PU axis to lift
    mAckError();
    fB_Axis.fI_TargetPosition := (fI_PositionClean1 / 1000);
    fB_Axis.fI_SpeedLimit     := sI_SpeedDef.fP_PlaceSpeed / 1000;
    
    IF bL_InPosClean1 OR bL_HigherPosC1 THEN
      fB_Axis.bI_MoveEnable := FALSE;
      bL_Busy               := FALSE;
      bL_Ready              := TRUE;  //Operation complete
    ELSE
      fB_Axis.bI_MoveEnable := bL_SafeMovePos;
      bL_Busy               := TRUE;
    END_IF
    
	2,3,4: //End
		bL_Busy  := FALSE;		
    bL_Ready := TRUE;  //Operation complete

	ELSE
		bL_Busy  := FALSE;		
    bL_Ready := TRUE;  //Operation complete
END_CASE
END_METHOD

{attribute 'monitoring' := 'call'}
PROPERTY pHigherPosC1 : bool
GET
pHigherPosC1 := bL_HigherPosC1;
END_GET
END_PROPERTY

{attribute 'monitoring' := 'call'}
PROPERTY pHigherPosWait : bool
GET
pHigherPosWait := bL_HigherPosWait;
END_GET
END_PROPERTY

{attribute 'monitoring' := 'call'}
PROPERTY pInPosClean1 : bool
GET
pInPosClean1 := bL_InPosClean1;
END_GET
END_PROPERTY

{attribute 'monitoring' := 'call'}
PROPERTY pInPosClean2 : bool
GET
pInPosClean2 := bL_InPosClean2;
END_GET
END_PROPERTY

{attribute 'monitoring' := 'call'}
PROPERTY pInPosPrint : bool
GET
pInPosPrint := bL_InPosPrint;
END_GET
END_PROPERTY

{attribute 'monitoring' := 'call'}
PROPERTY pInPosService : bool
GET
pInPosService := bL_InPosService;
END_GET
END_PROPERTY

{attribute 'monitoring' := 'call'}
PROPERTY pInPosWait : bool
GET
pInPosWait := bL_InPosWait;
END_GET
END_PROPERTY

PROPERTY pPositionPrint : REAL
GET
pPositionPrint := fI_PositionPrint;
END_GET
SET
fI_PositionPrint := pPositionPrint;
END_SET
END_PROPERTY

END_FUNCTION_BLOCK

// ---- POUs/Products/Machine/CleaningStation/FB_Cleaning_ValvePump.TcPOU
FUNCTION_BLOCK FB_Cleaning_ValvePump EXTENDS FB_CleanDevice
VAR_INPUT
END_VAR

VAR_OUTPUT
  bO_VacuumValve                  AT %Q* : BOOL;     (*Enable vacuum valve for CleaningStation*)

  bO_VacuumPump                   AT %Q* : BOOL;     (*Enable vacuum pump for CleaningStation*)
  wO_SetPointVacuumPump           AT %Q* : WORD;     (*Vacuum pump set point*)

  bO_CleanerPump                  AT %Q* : BOOL;     (*Enable cleaner pump for CleaningStation*)
  wO_SetPointCleanerPump          AT %Q* : WORD;     (*Cleaner pump set point*)
END_VAR

VAR
  _bManuEmptyTub                         : BOOL;     (*Manually empty tub*)

  bL_VacuumValve                         : BOOL;     (*Enable vacuum valve for CleaningStation*)

  bL_VacuumPump                          : BOOL;     (*Enable vacuum pump for CleaningStation*)
  lL_SetPointVacuumPump                  : DINT;     (*Vacuum pump set point [%]*)

  bL_CleanerPump                         : BOOL;     (*Enable cleaner pump for CleaningStation*)
  lL_SetPointCleanerPump                 : DINT;     (*Cleaner pump set point [%]*)

  fb_TonCleanerPumpOffset                : TON;
  fb_TonVacuumPumpDelay                  : TON;
END_VAR

VAR PERSISTENT
  lR_AnalogMaxDigitVacuumPump            : DINT := 16383;  (*Max value analog-output in digit (32767 = 10V)*)
  lR_SetPoint1VacuumPump                 : DINT;     (*Vacuum pump set point #1 [%]*)
  lR_SetPoint2VacuumPump                 : DINT;     (*Vacuum pump set point #2 [%]*)
  lR_SetPoint3VacuumPump                 : DINT;     (*Vacuum pump set point #3 [%]*)
  lR_SetPoint4VacuumPump                 : DINT;     (*Vacuum pump set point #4 [%]*)
  lR_AnalogMaxDigitCleanerPump           : DINT := 16383;  (*Max value analog-output in digit (32767 = 10V)*)
  lR_SetPoint1CleanerPump                : DINT;     (*Cleaner pump set point #1 [%]*)
  lR_SetPoint2CleanerPump                : DINT;     (*Cleaner pump set point #2 [%]*)
  lR_SetPoint3CleanerPump                : DINT;     (*Cleaner pump set point #3 [%]*)
  lR_SetPoint4CleanerPump                : DINT;     (*Cleaner pump set point #4 [%]*)

  tR_CleanerPumpOffset                   : TIME := T#4S;
  tR_VacuumPumpDelay                     : TIME := T#1S;
  tR_VacuumPumpEmptyBin                  : TIME := T#15S;
END_VAR

METHOD mCleaning : BOOL
VAR_INPUT
  iI_Step : INT;
END_VAR
//Abort: Stop pumps and return
IF bL_AbortReq THEN
  bL_Busy        := FALSE;
  bL_Ready       := TRUE;
  bL_VacuumValve := FALSE;
  bL_VacuumPump  := FALSE;
  bL_CleanerPump := FALSE;
  mSetOutput();
  RETURN;
END_IF

//Normal operation
CASE iI_Step OF
  0: //Init - Check if axis is not activated, restore safety
    fb_TonCleanerPumpOffset(IN := FALSE, PT := tR_CleanerPumpOffset);
    fb_TonVacuumPumpDelay  (IN := FALSE, PT := tR_VacuumPumpDelay);

    bL_Busy := FALSE;

  1: //Wait for PU axis to lift
    bL_Busy := FALSE;
    
  2: //Wait for CU axis to move out
    bL_Busy := FALSE;
    
  3: //Wait for PU axis to lower
    bL_Busy := FALSE;
    
  4: //Ensure CH axis is at starting position
    bL_Busy := FALSE;

  5: //Move CH to clean start position
    bL_Busy := FALSE;

  6: //Wait until cleaning equipment ready
    bL_VacuumValve         := TRUE;

    bL_VacuumPump          := TRUE;
    lL_SetPointVacuumPump  := lR_SetPoint1VacuumPump;

    bL_CleanerPump         := TRUE;
    lL_SetPointCleanerPump := lR_SetPoint1CleanerPump;
    
    mSetOutput();

    (*Delay cleaner pump for a good start-up.*)
    fb_TonCleanerPumpOffset(IN := TRUE, PT := tR_CleanerPumpOffset);
    bL_Busy := NOT fb_TonCleanerPumpOffset.Q;
    
  7: //Cleaning
    bL_Busy := FALSE;
    
  8: //Wait until cleaning equipment ready
    bL_VacuumValve         := TRUE;

    bL_VacuumPump          := TRUE;
    lL_SetPointVacuumPump  := lR_SetPoint1VacuumPump;

    bL_CleanerPump         := FALSE;
    lL_SetPointCleanerPump := lR_SetPoint1CleanerPump;
    
    mSetOutput();

    bL_Busy := FALSE;
    
  9: //Move CH to end position
    (*Off delay vacuum pump.*)
    fb_TonVacuumPumpDelay(IN := TRUE, PT := tR_VacuumPumpDelay);
    bL_Busy := NOT fb_TonVacuumPumpDelay.Q;
    
  10: //Wait for PU axis to lift
    bL_VacuumValve := FALSE;
    bL_VacuumPump  := FALSE;
    mSetOutput();

    bL_Busy := FALSE;
    
  11: //Move CH back to start 
    bL_VacuumValve         := FALSE;

    bL_VacuumPump          := TRUE;
    lL_SetPointVacuumPump  := lR_SetPoint1VacuumPump;

    bL_CleanerPump         := FALSE;
    lL_SetPointCleanerPump := lR_SetPoint1CleanerPump;
    
    mSetOutput();

    bL_Busy := FALSE;
    
  12: //End
    bL_VacuumValve := FALSE;
    bL_VacuumPump  := FALSE;
    mSetOutput();

    bL_Busy := FALSE;
  
  ELSE
    bL_Busy := FALSE;    
END_CASE
END_METHOD

METHOD mManuSetCleanerPump
VAR_INPUT
  bI_CleanerPump                         : BOOL;     (*Enable cleaner pump for CleaningStation*)
  bI_VacuumPump                          : BOOL;     (*Enable vacuum pump for CleaningStation*)
  wI_SetPointCleanerPump                 : DINT;     (*Cleaner pump set point*)
END_VAR
IF bI_CleanerPump THEN
  bO_CleanerPump         := TRUE;
  wO_SetPointCleanerPump := DINT_TO_WORD(lR_AnalogMaxDigitCleanerPump * wI_SetPointCleanerPump / 100);

  bO_VacuumPump          := bI_VacuumPump;                                                              
  wO_SetPointVacuumPump  := DINT_TO_WORD(lR_AnalogMaxDigitVacuumPump);
ELSE
  bO_CleanerPump         := FALSE;
  bO_VacuumPump          := FALSE;
END_IF
END_METHOD

METHOD mProduction : BOOL
VAR_INPUT
  iI_Step : INT;
END_VAR
//Abort: Stop whereever axis is and return
IF bL_AbortReq THEN
  bL_Busy        := FALSE;
  bL_Ready       := TRUE;
  bL_VacuumValve := FALSE;
  bL_VacuumPump  := FALSE;
  bL_CleanerPump := FALSE;
  mSetOutput();
  RETURN;
END_IF

//Normal operation
CASE iI_Step OF
  0: //Init - Check if axis is not activated, restore safety
    fb_TonCleanerPumpOffset(IN := FALSE, PT := tR_VacuumPumpEmptyBin);

    bL_Busy := FALSE;

  1: //Wait for PU axis to lift
    bL_Busy := FALSE;
    
  2: //Wait for CU axis to move out & empty bin
    (*Timer vacuum pump to empty bin.*)
    fb_TonCleanerPumpOffset(IN := TRUE, PT := tR_VacuumPumpEmptyBin);

    bL_VacuumValve         := FALSE;

    bL_VacuumPump          := NOT fb_TonCleanerPumpOffset.Q;
    lL_SetPointVacuumPump  := lR_SetPoint1VacuumPump;

    mSetOutput();

    bL_Busy := FALSE;
    
  3: //Wait for PU axis to lower
    (*Timer vacuum pump to empty bin.*)
    fb_TonCleanerPumpOffset(IN := TRUE, PT := tR_VacuumPumpEmptyBin);

    bL_VacuumValve := FALSE;
    bL_VacuumPump  := NOT fb_TonCleanerPumpOffset.Q;
    mSetOutput();

    bL_Busy := NOT fb_TonCleanerPumpOffset.Q;
    
  4: //End
    bL_VacuumValve := FALSE;
    bL_VacuumPump  := FALSE;
    mSetOutput();

    bL_Busy := FALSE;

  ELSE
    bL_Busy := FALSE;    
END_CASE
END_METHOD

METHOD mSetOutput
VAR_INPUT
END_VAR
bO_VacuumValve         := bL_VacuumValve;

bO_VacuumPump          := bL_VacuumPump;
wO_SetPointVacuumPump  := DINT_TO_WORD(lR_AnalogMaxDigitVacuumPump * lL_SetPointVacuumPump / 100);

bO_CleanerPump         := bL_CleanerPump;
wO_SetPointCleanerPump := DINT_TO_WORD(lR_AnalogMaxDigitCleanerPump * lL_SetPointCleanerPump / 100);
END_METHOD

PROPERTY pManuEmptyTub : BOOL
GET
pManuEmptyTub := _bManuEmptyTub;
END_GET
SET
_bManuEmptyTub := pManuEmptyTub;
IF _bManuEmptyTub THEN
  bO_VacuumValve         := FALSE;
  bO_VacuumPump          := TRUE;
  wO_SetPointVacuumPump  := DINT_TO_WORD(lR_AnalogMaxDigitVacuumPump);
ELSE
  bO_VacuumValve         := FALSE;
  bO_VacuumPump          := FALSE;
END_IF
END_SET
END_PROPERTY

END_FUNCTION_BLOCK

// ---- POUs/Products/FB_MOTION_INTERLOCK.TcPOU
FUNCTION_BLOCK FB_MOTION_INTERLOCK
(******************************************************************************************)
(*	FILENAME:	FB_MOTION_INTERLOCK								*)
(*	PROJECT:	Steinemann												*)
(*	COPYRIGHT:	Wifag-Polytype									*)
(*	ENVIRONMENT:	TwinCat2, v2.11								*)
(*	VERSION:	1.0																*)
(*	DESCRIPTION:																*)
(*		Interlock for X,Y and Z axis					 		*)
(*	AUTHOR:	FAF																	*)
(*																*)
(******************************************************************************************)
(*	Changes:													*)
(******************************************************************************************)
(*	Date	Authtor	Descriptons																															*)
(******************************************************************************************)
VAR_INPUT
	fICU_Position	: REAL;		(*X: Cleaning Unit Position*)
	fIPU_Position	: REAL;		(*Z: Print Unit Position*)
	bICU_PositionUnknown : BOOL:=TRUE;	(*X: Position Unknown*)
	bIPU_PositionUnknown : BOOL:=TRUE;	(*Z: Position Unknown*)

	fCCU_Tolerance		: REAL:=0.001;				 (*CU Positioning Tolerance*)
	fCPU_Tolerance		: REAL:=0.0005;				 (*PU Positioning Tolerance*)
	fCCU_SafePosition	: ARRAY[1..3] OF REAL; (*Safe Operating Area from -INF to this value*)
	fCPU_SafePosition	: ARRAY[1..2] OF REAL; (*Safe Operating Area from this Value to +INF*)
	fCCU_CleaningPosition	: REAL;
END_VAR

VAR_OUTPUT
	bOPU_MoveAuth	: BOOL;	(*Move authorized*)
	bOCU_MoveAuth	: BOOL;	(*Move authorized*)
	bOCH_MoveAuth	: BOOL;	(*Move authorized*)
	bO_InterlockActive : BOOL;
END_VAR
VAR
END_VAR

(*Print Unit Interlock ----------------------------------------------------------------*)
IF fICU_Position < fCCU_SafePosition[1] + fCCU_Tolerance THEN		(*Cleaning Unit not in collision area*)
	bOPU_MoveAuth:=TRUE;

//ELSIF fICU_Position < fCCU_SafePosition[2] - fCCU_Tolerance THEN	(*Cleaning Unit in collision area*)
ELSIF fICU_Position < fCCU_CleaningPosition - fCCU_Tolerance THEN	(*Cleaning Unit in collision area*)
	IF fIPU_Position > fCPU_SafePosition[2] THEN
		bOPU_MoveAuth:=TRUE;
	ELSE
		bOPU_MoveAuth:=FALSE;
	END_IF;

ELSIF fICU_Position < fCCU_SafePosition[3] + fCCU_Tolerance THEN	(*Cleaning Unit in Cleaning Position*)
	IF fIPU_Position > fCPU_SafePosition[1] THEN
		bOPU_MoveAuth:=TRUE;
	ELSE
		bOPU_MoveAuth:=FALSE;
	END_IF;

ELSE																						(*Cleaning Unit in collision area*)
	IF fIPU_Position > fCPU_SafePosition[2] THEN
		bOPU_MoveAuth:=TRUE;
	ELSE
		bOPU_MoveAuth:=FALSE;
	END_IF;
END_IF;

IF bICU_PositionUnknown THEN	(*No movement allowed when X-Pos unknown*)
	bOPU_MoveAuth:=FALSE;
END_IF;

(*Clean Unit/Head Interlock ----------------------------------------------------------------*)

IF fICU_Position < fCCU_SafePosition[1] THEN		(*Cleaning Unit not in collision area*)
	bOCU_MoveAuth:=TRUE;
	bOCH_MoveAuth:=TRUE;

//ELSIF fICU_Position < fCCU_SafePosition[2] THEN	(*Cleaning Unit in collision area*)
ELSIF fICU_Position < fCCU_CleaningPosition - fCCU_Tolerance THEN	(*Cleaning Unit in collision area*)
	IF fIPU_Position > fCPU_SafePosition[2]-fCPU_Tolerance THEN
		bOCU_MoveAuth:=TRUE;
		bOCH_MoveAuth:=TRUE;
	ELSE
		bOCU_MoveAuth:=FALSE;
    IF fICU_Position = fCCU_SafePosition[1] THEN		(*Cleaning outside of machine*)
		  bOCH_MoveAuth:=TRUE;
    ELSE
		  bOCH_MoveAuth:=FALSE;
    END_IF;
  END_IF;

ELSIF fICU_Position < fCCU_SafePosition[3] + fCCU_Tolerance THEN	(*Cleaning Unit in Cleaning Position*)
	IF fIPU_Position > fCPU_SafePosition[2] - fCPU_Tolerance THEN
		bOCU_MoveAuth:=TRUE;
	ELSE
		bOCU_MoveAuth:=FALSE;
	END_IF;

	(*CU must be in Cleaning Position for the CH to move*)
	IF ABS(fCCU_CleaningPosition - fICU_Position) < 2*fCCU_Tolerance THEN
		bOCH_MoveAuth:=TRUE;
	ELSE

//		IF fIPU_Position > fCPU_SafePosition[2] - fCPU_Tolerance THEN
//			bOCH_MoveAuth:=TRUE;
//		ELSE
//			bOCH_MoveAuth:=FALSE;
//		END_IF;
	END_IF;

ELSE																						(*Cleaning Unit in collision area*)
	IF fIPU_Position > fCPU_SafePosition[2] - fCPU_Tolerance THEN
		bOCU_MoveAuth:=TRUE;
		bOCH_MoveAuth:=TRUE;
	ELSE
		bOCU_MoveAuth:=FALSE;
		bOCH_MoveAuth:=FALSE;
	END_IF;
END_IF;

IF (bICU_PositionUnknown AND (fIPU_Position < (fCPU_SafePosition[2] - fCPU_Tolerance))) OR bIPU_PositionUnknown THEN	(*No movement allowed when X-Pos unknown*)
	bOCU_MoveAuth:=FALSE;
	bOCH_MoveAuth:=FALSE;
END_IF;



bO_InterlockActive:=NOT(bOCU_MoveAuth AND bOPU_MoveAuth AND bOCH_MoveAuth);

END_FUNCTION_BLOCK

// ---- POUs/Products/FB_MOTION_TO_INKSYSTEM_IF.TcPOU
FUNCTION_BLOCK FB_MOTION_TO_INKSYSTEM_IF
(******************************************************************************************)
(*	FILENAME:	FB_MOTION_TO_INKSYSTEM_IF							*)
(*	PROJECT:	Steinemann										*)
(*	COPYRIGHT:	Wifag-Polytype									*)
(*	ENVIRONMENT:	TwinCat2, v2.11								*)
(*	VERSION:	1.0												*)
(*	DESCRIPTION:												*)
(*		Interface block to link ink to motion system		*)
(*	AUTHOR:	FAF							*)
(*																*)
(******************************************************************************************)
(*	Changes:													*)
(******************************************************************************************)
(*	Date	Authtor	Descriptons									*)
(*																*)
(******************************************************************************************)
VAR_INPUT
	(*Commands from Cleaning Process Controller*)
	sI_CleanDevCmd				: ST_CLEANING_DEV_CMD;	(*Initialize operation*)

	(*Inputs from Purge Controller*)
	bI_PurgeBusy					: BOOL;
	bI_CleanPumpOn				: BOOL;
END_VAR
VAR_OUTPUT
	(*To machine/user*)
	sO_CleanDevStatus			:ST_CLEANING_DEV_STATUS;	(*Initialize operation*)
	bO_Purge							: BOOL;
	bO_EnableCleanerPump	: BOOL;
END_VAR
VAR
	bL_PurgeStarted				: BOOL;
	TonDelay							: TON;									(*Time wait for intertask comm*)
END_VAR

(*Mode selection*)
IF sI_CleanDevCmd.bAuto THEN	(*Control by cleaning process*)
	CASE 	sI_CleanDevCmd.eOperation OF
		eNOP:	(*No operation active*)
			bO_Purge :=	FALSE;
			bL_PurgeStarted:=FALSE;
			bO_EnableCleanerPump := FALSE;
			TonDelay.IN:= FALSE;

		eOPCLEAN:	(*Cleaning Mode -------------------------------------*)
			bO_Purge :=	FALSE;
			bL_PurgeStarted:=FALSE;
			IF sI_CleanDevCmd.bInit THEN
				bO_EnableCleanerPump := FALSE;
			ELSIF sI_CleanDevCmd.bPrep THEN
				bO_EnableCleanerPump := FALSE;
			ELSIF sI_CleanDevCmd.bStart THEN
				bO_EnableCleanerPump := TRUE;
			ELSIF sI_CleanDevCmd.bStop THEN
				bO_EnableCleanerPump := FALSE;
			ELSE	(*Command removed, wait until axis finished movement*)
				;		(*No operation, keep commands*)
			END_IF;

			TonDelay.PT:= T#500ms;
			TonDelay.IN:= bO_EnableCleanerPump;
			TonDelay();

			IF bO_EnableCleanerPump THEN
				sO_CleanDevStatus.bBusy:=NOT(TonDelay.Q AND bI_CleanPumpOn);
				sO_CleanDevStatus.bReady:=TonDelay.Q AND bI_CleanPumpOn;
			ELSE
				sO_CleanDevStatus.bBusy:=FALSE;
				sO_CleanDevStatus.bReady:=TRUE;
			END_IF;

			sO_CleanDevStatus.bBusy:= (bO_EnableCleanerPump AND NOT bI_CleanPumpOn) OR (NOT bO_EnableCleanerPump AND bI_CleanPumpOn);
			sO_CleanDevStatus.bReady:= NOT sO_CleanDevStatus.bBusy;

		eOPPURGE:	(*Purge Mode -------------------------------------*)
			bO_EnableCleanerPump :=	FALSE;
			IF sI_CleanDevCmd.bInit THEN
				bO_Purge := FALSE;
			ELSIF sI_CleanDevCmd.bPrep THEN
				bO_Purge := FALSE;
			ELSIF sI_CleanDevCmd.bStart THEN
				bO_Purge := TRUE;
			ELSIF sI_CleanDevCmd.bStop THEN
				bO_Purge := FALSE;
			ELSE	(*Command removed, wait until axis finished movement*)
				;		(*No operation, keep commands*)
			END_IF;

			IF bO_Purge THEN
					IF bI_PurgeBusy THEN
						bL_PurgeStarted:=TRUE;
					END_IF;
					sO_CleanDevStatus.bBusy:= NOT(bL_PurgeStarted AND NOT bI_PurgeBusy);
					sO_CleanDevStatus.bReady:= bL_PurgeStarted AND NOT bI_PurgeBusy;
			ELSE
				bL_PurgeStarted:=FALSE;
				sO_CleanDevStatus.bBusy:=FALSE;
				sO_CleanDevStatus.bReady:=TRUE;
			END_IF;

		ELSE
				TonDelay.IN:= FALSE;
				bO_Purge :=	FALSE;
				bL_PurgeStarted:=FALSE;
				bO_EnableCleanerPump := FALSE;
				sO_CleanDevStatus.bBusy:=FALSE;
				sO_CleanDevStatus.bReady:=TRUE;
		END_CASE;
END_IF;

IF sI_CleanDevCmd.bAbort THEN
		TonDelay.IN:= FALSE;
		bO_Purge :=	FALSE;
		bL_PurgeStarted:=FALSE;
		bO_EnableCleanerPump := FALSE;
		sO_CleanDevStatus.bBusy:=FALSE;
		sO_CleanDevStatus.bReady:=TRUE;
END_IF;

sO_CleanDevStatus.bRefKnown:=TRUE;

END_FUNCTION_BLOCK

// ---- POUs/Products/Machine/FB_CappingCommand.TcPOU
FUNCTION_BLOCK FB_CappingCommand

VAR_INPUT
  IbTrigger                                 : BOOL;
  IbReset                                   : BOOL;
END_VAR

VAR_OUTPUT
  ObCappingCommand                          : BOOL;
END_VAR

VAR
  fb_TonTrigger                             : TON;
  fb_TonReset                               : TON;
  bL_CappingCommandAfterEngaged             : BOOL;
END_VAR

VAR CONSTANT
  tC_DELAY_CAPPING_COMMAND                  : TIME := T#500MS;    (*Delay for automatic generated capping commands*)
  tC_RELEASE_CAPPING_COMMAND                : TIME := T#2S;       (*Release for automatic generated capping commands*)
END_VAR

fb_TonTrigger(IN := IbTrigger, PT := tC_DELAY_CAPPING_COMMAND);
IF fb_TonTrigger.Q THEN
  ObCappingCommand := TRUE;
END_IF
fb_TonReset(IN := IbTrigger, PT := tC_RELEASE_CAPPING_COMMAND);
IF fb_TonReset.Q OR IbReset THEN
  ObCappingCommand := FALSE;
END_IF

END_FUNCTION_BLOCK

// ---- POUs/Projects/Machine/FB_MachineComm.TcPOU
FUNCTION_BLOCK FB_MachineComm EXTENDS FB_Sim
VAR_INPUT
  // from prg internals to machine
  sModuleMachineFeedback : ARRAY[1..iCPr_NB_PM] OF ST_ModuleMachineInterface_OUT;
END_VAR
VAR_OUTPUT
  // from machine -> prg internals
  sModuleMachineState : ARRAY[1..iCPr_NB_PM] OF ST_ModuleMachineInterface_IN;
END_VAR
VAR
  bInit : BOOL;
  nCtr : UDINT;
  _bSimOk : BOOL;
  _bSimRand : BOOL;
  _fMaxSpeed : LREAL;       // max. speed over all modules
  _bSpeedExeeded : BOOL;    // one module exceeded speed
  _bMachineMoving : BOOL;   // one module is moving
  
  // view
  nSelPm : UDINT := 1;     // selected pm in view
END_VAR

IF NOT bInit THEN Init(); RETURN; END_IF
SUPER^();

// TODO: move all EAP or handling structure to this fb

FOR nCtr := 1 TO TO_UDINT(iCPr_NB_PM) DO 
  {warning 'TODO: SubstrateLength from Job or Machine? Check somewhere'}  
  sModuleMachineState[nCtr].bEStop                 := getValueBool ( PRG_MACHINE.iSystemStatus.bEmergency, FALSE);
  sModuleMachineState[nCtr].bSleep                 := getValueBool ( PRG_MACHINE.iSystemStatus.bSleep, FALSE);
  sModuleMachineState[nCtr].bSafetyCoverOk         := getValueBool ( PRG_MACHINE.bIKp_SafetyCoverOK[nCtr], TRUE);
  sModuleMachineState[nCtr].bServiceDoorsOk        := getValueBool ( PRG_MACHINE.bIKp_SafetyDoorsOK[nCtr], TRUE);
  sModuleMachineState[nCtr].bExhaustVacuumWarning  := getValueBool ( PRG_MACHINE.fb_ExhaustSystem[nCtr].bO_VacuumWarningLevel, FALSE);
  sModuleMachineState[nCtr].bExhaustVacuumError    := getValueBool ( PRG_MACHINE.fb_ExhaustSystem[nCtr].bO_VacuumErrorLevel, FALSE);
  sModuleMachineState[nCtr].bExhaustFUError        := getValueBool ( FALSE, FALSE); // NOT fb_ExhaustSystem[1].bO_FURead
  sModuleMachineState[nCtr].bDriftControlError     := getValueBool ( FALSE, FALSE); // fB_DriftControl[nCtr].bO_SupervisionContrErr OR fB_DriftControl[nCtr].bO_ContrErr
  sModuleMachineState[nCtr].bDriftControlMissMarks := getValueBool ( FALSE, FALSE); // fB_DriftControl[nCtr].bO_SupervisionMissMarks
  sModuleMachineState[nCtr].bSafetyOk              := getValueBool ( PRG_MACHINE.bL_SafetyOk[nCtr], TRUE);
  sModuleMachineState[nCtr].bUnitInPrintPosition   := getValueBool ( PRG_MACHINE.fb_CleaningPU[nCtr].pInPosPrint, TRUE);
  sModuleMachineState[nCtr].bEngaged               := getValueBool ( PRG_MACHINE.bL_IO_Engaged[nCtr] OR PRG_MACHINE.bSimulation, TRUE);
  sModuleMachineState[nCtr].bPrintEnabled          := getValueBool ( (PRG_MACHINE.IbEAP_PrintEnabled[nCtr] AND PRG_MACHINE.fb_CleaningPU[nCtr].pInPosPrint) OR PRG_MACHINE.bSimulation, TRUE);
  sModuleMachineState[nCtr].fSubstrateThickness    := getValueLreal( TO_LREAL(PRG_MACHINE.InEAP_SubstrateThickness) / 1_000_000, 0.003);    (*[µm] => [m]*)
  sModuleMachineState[nCtr].fSubstrateLen          := getValueLreal( TO_LREAL(PRG_MACHINE.InEAP_FormatLength) / 1_000_000, 0.55);    (*[µm] => [m]*) 
  sModuleMachineState[nCtr].fWebStretchCalculated  := getValueLreal( (1.0 - (DINT_TO_LREAL(PRG_MACHINE.InEAP_WebStretchFactor) / 1_000_000)), 0.99);
  sModuleMachineState[nCtr].fLateralRegister       := getValueLreal( TO_LREAL(PRG_MACHINE.InEAP_LateralRegister) / 1_000_000, 0);
  sModuleMachineState[nCtr].fModule2ToModule3      := getValueLreal( TO_LREAL(PRG_MACHINE.InEAP_Module2ToModule3) / 1_000_000, 4.5);
  sModuleMachineState[nCtr].bTargetSpeedReached    := getValueBool (  PRG_MACHINE.IbEAP_TargetSpeedReached, TRUE);
  sModuleMachineState[nCtr].fNeutralFibreFactor    := getValueLreal( TO_LREAL(PRG_MACHINE.InEAP_NeutralFibreFactor), 98);
END_FOR


// get global values over all modules
_fMaxSpeed := getMaxSpeed();
_bSpeedExeeded := _bMachineMoving := FALSE;
FOR nCtr := 1 TO TO_UDINT(iCPr_NB_PM) DO
  _bSpeedExeeded := _bSpeedExeeded OR sModuleMachineFeedback[nCtr].bSpeedExeeded;
  _bMachineMoving := _bMachineMoving OR sModuleMachineFeedback[nCtr].bMoving;
END_FOR

// simulation
IF bSimEnable THEN
  IF    _nModeSel = 1 THEN _bSimOk := TRUE;  _bSimRand := FALSE;
  ELSIF _nModeSel = 2 THEN _bSimOk := FALSE; _bSimRand := TRUE;
  END_IF
ELSE
  _bSimOk := FALSE;
  _bSimRand := FALSE;
END_IF

PROPERTY bMachineMoving : BOOL
GET
bMachineMoving := _bMachineMoving;
END_GET
END_PROPERTY

PROPERTY bSpeedExeeded : BOOL
GET
VAR
  i : UDINT;
END_VAR
bSpeedExeeded := _bSpeedExeeded;
END_GET
END_PROPERTY

METHOD PRIVATE getMaxSpeed : LREAL
VAR
  f : LREAL;
  i : UDINT;
END_VAR
f := 0;
FOR i:=1 TO TO_UDINT(iCPr_NB_PM) DO
  IF sModuleMachineFeedback[i].fMaxSpeed = 0 THEN
    ; // invalid speed
  ELSIF f = 0 OR f > sModuleMachineFeedback[i].fMaxSpeed THEN
    f := sModuleMachineFeedback[i].fMaxSpeed;
	END_IF
END_FOR

getMaxSpeed := f;
END_METHOD

METHOD PRIVATE getValueBool : BOOL
VAR_INPUT
  in   : BOOL;   // input value
  sim  : BOOL;   // default simulation value - ok state
END_VAR
VAR_INST
  rand : DRAND := (Seed:=14);
END_VAR
rand();
IF    _bSimOk   THEN getValueBool := sim;
ELSIF _bSimRand THEN getValueBool := SEL(rand.Num > 0.5, FALSE, TRUE);
ELSE                 getValueBool := in;
END_IF
END_METHOD

METHOD PRIVATE getValueLreal : LREAL
VAR_INPUT
  in   : LREAL;   // input value
  sim  : LREAL;   // default simulation value - ok state
END_VAR
VAR_INST
  rand : DRAND := (Seed:=14);
  randFactor : LREAL := 10;
END_VAR
rand();
IF    _bSimOk   THEN getValueLreal := sim;
ELSIF _bSimRand THEN getValueLreal := rand.Num * randFactor;
ELSE                 getValueLreal := in;
END_IF
END_METHOD

METHOD Init : BOOL
VAR
  sMode : ST_SimModeDef;
END_VAR
(*
sMode.aMode := 'default';  // sim ok
sMode.sCfg := '{ "desc":"sim machine all ok inputs" }';
setMode(sMode:=sMode);
*)
sMode.aMode := 'sim random';
sMode.sCfg := '{ "desc":"sim random inpus" }';
setMode(sMode:=sMode);

bInit := TRUE;
END_METHOD

(*Max. possible speed [m/min]*)
PROPERTY nMaxSpeedMpMin : DINT
GET
nMaxSpeedMpMin := TO_DINT(_fMaxSpeed * 60);
END_GET
END_PROPERTY

END_FUNCTION_BLOCK

// ---- POUs/Products/Machine/FB_ExhaustSystemPrint.TcPOU
FUNCTION_BLOCK FB_ExhaustSystemPrint

VAR_INPUT
  bI_FUReady                         AT %I* : BOOL;   (*FU ready*)
  iI_VacuumMeasurement               AT %I* : UINT;   (*Analog input: vacuum measurement*)
  bI_AerosolMeasurementAckInit       AT %I* : BOOL;                  (*EL6001: aerosol measurement acknowledge init*)
  bI_AerosolMeasurementDataRec       AT %I* : BOOL;                  (*EL6001: aerosol measurement receive data*)
  iI_AerosolMeasurementRecDataLength AT %I* : USINT;                 (*EL6001: aerosol measurement receive data length*)
  cI_AerosolMeasurementRxBuff        AT %I* : ARRAY[0..21] OF BYTE;  (*EL6001: aerosol measurement receive data buffer*)
  bI_AerosolMeasurementBufferFull    AT %I* : BOOL;                  (*EL6001: aerosol measurement buffer full*)
  bI_AerosolMeasurementFramingError  AT %I* : BOOL;                  (*EL6001: aerosol measurement framing error*)
  bI_AerosolMeasurementOverRunError  AT %I* : BOOL;                  (*EL6001: aerosol measurement over run error*)

  bI_PrintActive                            : BOOL;   (*Printing active*)
END_VAR

VAR_OUTPUT
  bO_FUActivate                      AT %Q* : BOOL;   (*FU activation*)
  bO_AerosolMeasurementReqInit       AT %Q* : BOOL;   (*EL6001: aerosol measurement request init*)
  bO_AerosolMeasurementAckRec        AT %Q* : BOOL;   (*EL6001: aerosol measurement acknowledge receive*)

  bO_FUReady                                : BOOL;   (*FU ready*)
  bO_VacuumWarningLevel                     : BOOL;   (*Vacuum warning level reached*)
  bO_VacuumErrorLevel                       : BOOL;   (*Vacuum error level reached*)
END_VAR

VAR
  iL_Counter                                : INT;    (*Basic counter*)

  fb_TofFUOffDelay                          : TOF;    (*FU off delay*)
  fb_TonVacuumCheckDelay                    : TON;    (*Vacuum check delay*)

  fL_VacuumAnalogLevelMBar                  : REAL;   (*Actual value analog-input in mBar*)

  (*Aerosol measurement*)
  fb_TonMeasurementTrigger                  : TON;                   (*Vacuum check delay*)
  eO_ComState                               : EN_COMPORT_STATES;     (*State of the COM port*)
  iL_ComState                               : INT := 0;              (*Identifier on the state of the com function*)
  cL_Value                                  : BYTE;                  (*Amount of data received*)
  aL_ReceivedData                           : T_MaxString;           (*String for received data*)
  fb_RTrigDataReceived                      : R_TRIG;                (*R_TRIG for data received*)
  fb_FTrigDataReceived                      : F_TRIG;                (*F_TRIG for data received*)
  iL_ReceiveCount                           : UINT;                  (*Receive counter*)
  fL_ParticleMeasurements                   : ARRAY[1..iC_ParticleMeasurementNb] OF REAL;  (*Particle measurements*)
  iL_ParticleMeasurementIdx                 : INT := 1;              (*Particle measurement index*)
END_VAR

VAR PERSISTENT
  tR_FUOffDelay                             : TIME := T#3M;   (*FU off delay time*)
  tR_VacuumCheckDelay                       : TIME := T#10S;  (*Vacuum check delay time*)

